LIN {X 0,Y 125.443,Z 652.418,A -85,B 0,C 180,E1 -25686.032,E2 -25686.032} C_VEL
LIN {X 0,Y 130.254,Z 643.589,A -85,B 0,C 180,E1 -25690.349,E2 -25690.349} C_VEL
LIN {X 0,Y 135.865,Z 633.156,A -85,B 0,C 180,E1 -25694.291,E2 -25694.291} C_VEL
LIN {X 0,Y 142.077,Z 620.726,A -85,B 0,C 180,E1 -25697.899,E2 -25697.899} C_VEL
LIN {X 0,Y 147.675,Z 608.285,A -85,B 0,C 180,E1 -25700.654,E2 -25700.654} C_VEL
LIN {X 0,Y 152.859,Z 595.068,A -85,B 0,C 180,E1 -25702.913,E2 -25702.913} C_VEL
LIN {X 0,Y 157.703,Z 580.518,A -85,B 0,C 180,E1 -25704.803,E2 -25704.803} C_VEL
LIN {X 0,Y 161.766,Z 565.791,A -85,B 0,C 180,E1 -25706.188,E2 -25706.188} C_VEL
LIN {X 0,Y 165,Z 549.941,A -85,B 0,C 180,E1 -25707.268,E2 -25707.268} C_VEL
LIN {X 0,Y 167.218,Z 532.789,A -85,B 0,C 180,E1 -25708.056,E2 -25708.056} C_VEL
LIN {X 0,Y 172.706,Z 478.21,A -85,B 0,C 180,E1 -25710.075,E2 -25710.075} C_VEL
LIN {X 0,Y 167.716,Z 464.569,A -85,B 0,C 180,E1 -25713.059,E2 -25713.059} C_VEL
LIN {X 0,Y 162.081,Z 450.718,A -85,B 0,C 180,E1 -25716.721,E2 -25716.721} C_VEL
LIN {X 0,Y 156.963,Z 439.698,A -85,B 0,C 180,E1 -25720.339,E2 -25720.339} C_VEL
LIN {X 0,Y 151.626,Z 431.129,A -85,B 0,C 180,E1 -25724.439,E2 -25724.439} C_VEL
LIN {X 0,Y 146.698,Z 423.586,A -85,B 0,C 180,E1 -25728.832,E2 -25728.832} C_VEL
LIN {X 0,Y 143.791,Z 419.372,A -85,B 0,C 180,E1 -25731.835,E2 -25731.835} C_VEL
LIN {X 0,Y 140.329,Z 414.378,A -85,B 0,C 180,E1 -25736.007,E2 -25736.007} C_VEL
LIN {X 0,Y 137.906,Z 411.663,A -85,B 0,C 180,E1 -25739.367,E2 -25739.367} C_VEL
LIN {X 0,Y 136.739,Z 409.178,A -85,B 0,C 180,E1 -25741.474,E2 -25741.474} C_VEL
LIN {X 0,Y 133.888,Z 406.923,A -85,B 0,C 180,E1 -25747.021,E2 -25747.021} C_VEL
LIN {X 0,Y 132.787,Z 404.232,A -85,B 0,C 180,E1 -25750.732,E2 -25750.732} C_VEL
LIN {X 0,Y 131.279,Z 403.638,A -85,B 0,C 180,E1 -25758.737,E2 -25758.737} C_VEL
LIN {X 0,Y 132.384,Z 404.128,A -85,B 0,C 180,E1 -25768.976,E2 -25768.976} C_VEL
LIN {X 0,Y 133.882,Z 407.624,A -85,B 0,C 180,E1 -25774.373,E2 -25774.373} C_VEL
LIN {X 0,Y 136.345,Z 409.759,A -85,B 0,C 180,E1 -25779.23,E2 -25779.23} C_VEL
LIN {X 0,Y 138.489,Z 413.228,A -85,B 0,C 180,E1 -25782.831,E2 -25782.831} C_VEL
LIN {X 0,Y 140.328,Z 415.144,A -85,B 0,C 180,E1 -25785.268,E2 -25785.268} C_VEL
LIN {X 0,Y 142.881,Z 418.739,A -85,B 0,C 180,E1 -25788.424,E2 -25788.424} C_VEL
LIN {X 0,Y 144.144,Z 420.426,A -85,B 0,C 180,E1 -25789.796,E2 -25789.796} C_VEL
LIN {X 0,Y 147.549,Z 425.18,A -85,B 0,C 180,E1 -25793.178,E2 -25793.178} C_VEL
LIN {X 0,Y 152.323,Z 432.249,A -85,B 0,C 180,E1 -25797.286,E2 -25797.286} C_VEL
LIN {X 0,Y 158.951,Z 442.925,A -85,B 0,C 180,E1 -25802.168,E2 -25802.168} C_VEL
LIN {X 0,Y 166.384,Z 455.969,A -85,B 0,C 180,E1 -25806.825,E2 -25806.825} C_VEL
LIN {X 0,Y 172.94,Z 469.275,A -85,B 0,C 180,E1 -25810.468,E2 -25810.468} C_VEL
LIN {X 0,Y 166.829,Z 528.834,A -85,B 0,C 180,E1 -25812.708,E2 -25812.708} C_VEL
LIN {X 0,Y 164.138,Z 544.967,A -85,B 0,C 180,E1 -25813.682,E2 -25813.682} C_VEL
LIN {X 0,Y 160.991,Z 559.376,A -85,B 0,C 180,E1 -25814.965,E2 -25814.965} C_VEL
LIN {X 0,Y 156.607,Z 574.603,A -85,B 0,C 180,E1 -25816.755,E2 -25816.755} C_VEL
LIN {X 0,Y 151.714,Z 588.809,A -85,B 0,C 180,E1 -25818.985,E2 -25818.985} C_VEL
LIN {X 0,Y 146.164,Z 602.31,A -85,B 0,C 180,E1 -25821.707,E2 -25821.707} C_VEL
LIN {X 0,Y 140.508,Z 614.537,A -85,B 0,C 180,E1 -25824.907,E2 -25824.907} C_VEL
LIN {X 0,Y 135.088,Z 625.294,A -85,B 0,C 180,E1 -25828.511,E2 -25828.511} C_VEL
LIN {X 0,Y 129.26,Z 635.988,A -85,B 0,C 180,E1 -25833.118,E2 -25833.118} C_VEL
LIN {X 0,Y 124.232,Z 644.963,A -85,B 0,C 180,E1 -25838.132,E2 -25838.132} C_VEL
LIN {X 0,Y 119.987,Z 652.541,A -85,B 0,C 180,E1 -25843.551,E2 -25843.551} C_VEL
LIN {X 0,Y 116.685,Z 658.822,A -85,B 0,C 180,E1 -25849.347,E2 -25849.347} C_VEL
LIN {X 0,Y 114.262,Z 664.018,A -85,B 0,C 180,E1 -25855.504,E2 -25855.504} C_VEL
LIN {X 0,Y 112.642,Z 668.237,A -85,B 0,C 180,E1 -25862.03,E2 -25862.03} C_VEL
LIN {X 0,Y 112.015,Z 671.471,A -85,B 0,C 180,E1 -25868.862,E2 -25868.862} C_VEL
LIN {X 0,Y 112.697,Z 673.827,A -85,B 0,C 180,E1 -25876.685,E2 -25876.685} C_VEL
LIN {X 0,Y 114.296,Z 674.743,A -85,B 0,C 180,E1 -25883.072,E2 -25883.072} C_VEL
LIN {X 0,Y 116.279,Z 674.886,A -85,B 0,C 180,E1 -25887.8,E2 -25887.8} C_VEL
LIN {X 0,Y 118.94,Z 674.527,A -85,B 0,C 180,E1 -25892.418,E2 -25892.418} C_VEL
LIN {X 0,Y 122.264,Z 673.586,A -85,B 0,C 180,E1 -25896.888,E2 -25896.888} C_VEL
LIN {X 0,Y 126.265,Z 672.105,A -85,B 0,C 180,E1 -25901.13,E2 -25901.13} C_VEL
LIN {X 0,Y 130.881,Z 670.075,A -85,B 0,C 180,E1 -25905.146,E2 -25905.146} C_VEL
LIN {X 0,Y 138.024,Z 666.375,A -85,B 0,C 180,E1 -25910.12,E2 -25910.12} C_VEL
LIN {X 0,Y 146.03,Z 661.626,A -85,B 0,C 180,E1 -25914.475,E2 -25914.475} C_VEL
LIN {X 0,Y 154.683,Z 655.759,A -85,B 0,C 180,E1 -25918.354,E2 -25918.354} C_VEL
LIN {X 0,Y 163.688,Z 648.719,A -85,B 0,C 180,E1 -25921.734,E2 -25921.734} C_VEL
LIN {X 0,Y 174.031,Z 639.5,A -85,B 0,C 180,E1 -25924.977,E2 -25924.977} C_VEL
LIN {X 0,Y 184.395,Z 628.842,A -85,B 0,C 180,E1 -25927.703,E2 -25927.703} C_VEL
LIN {X 0,Y 193.48,Z 617.944,A -85,B 0,C 180,E1 -25929.759,E2 -25929.759} C_VEL
LIN {X 0,Y 201.771,Z 606.367,A -85,B 0,C 180,E1 -25931.454,E2 -25931.454} C_VEL
LIN {X 0,Y 209.045,Z 594.538,A -85,B 0,C 180,E1 -25932.844,E2 -25932.844} C_VEL
LIN {X 0,Y 215.674,Z 581.801,A -85,B 0,C 180,E1 -25933.983,E2 -25933.983} C_VEL
LIN {X 0,Y 221.796,Z 567.365,A -85,B 0,C 180,E1 -25935.017,E2 -25935.017} C_VEL
LIN {X 0,Y 226.824,Z 552.153,A -85,B 0,C 180,E1 -25935.827,E2 -25935.827} C_VEL
LIN {X 0,Y 230.242,Z 538.347,A -85,B 0,C 180,E1 -25936.341,E2 -25936.341} C_VEL
LIN {X 0,Y 233.479,Z 518.913,A -85,B 0,C 180,E1 -25936.868,E2 -25936.868} C_VEL
LIN {X 0,Y 234.676,Z 510.745,A -85,B 0,C 180,E1 -25937.099,E2 -25937.099} C_VEL
LIN {X 0,Y 234.535,Z 509.573,A -85,B 0,C 180,E1 -25939.245,E2 -25939.245} C_VEL
LIN {X 0,Y 234.487,Z 510.416,A -85,B 0,C 180,E1 -25940.646,E2 -25940.646} C_VEL
LIN {X 0,Y 234.522,Z 512.099,A -85,B 0,C 180,E1 -25942.274,E2 -25942.274} C_VEL
LIN {X 0,Y 230.283,Z 538.9,A -85,B 0,C 180,E1 -25942.912,E2 -25942.912} C_VEL
LIN {X 0,Y 226.669,Z 553.893,A -85,B 0,C 180,E1 -25943.367,E2 -25943.367} C_VEL
LIN {X 0,Y 221.965,Z 568.306,A -85,B 0,C 180,E1 -25943.898,E2 -25943.898} C_VEL
LIN {X 0,Y 216.394,Z 581.875,A -85,B 0,C 180,E1 -25944.578,E2 -25944.578} C_VEL
LIN {X 0,Y 209.352,Z 595.9,A -85,B 0,C 180,E1 -25945.549,E2 -25945.549} C_VEL
LIN {X 0,Y 201.575,Z 608.795,A -85,B 0,C 180,E1 -25946.691,E2 -25946.691} C_VEL
LIN {X 0,Y 193.253,Z 620.7,A -85,B 0,C 180,E1 -25948.126,E2 -25948.126} C_VEL
LIN {X 0,Y 184.53,Z 631.604,A -85,B 0,C 180,E1 -25949.862,E2 -25949.862} C_VEL
LIN {X 0,Y 174.353,Z 642.657,A -85,B 0,C 180,E1 -25952.166,E2 -25952.166} C_VEL
LIN {X 0,Y 166.132,Z 650.629,A -85,B 0,C 180,E1 -25954.418,E2 -25954.418} C_VEL
LIN {X 0,Y 155.723,Z 659.68,A -85,B 0,C 180,E1 -25957.832,E2 -25957.832} C_VEL
LIN {X 0,Y 146.02,Z 667.142,A -85,B 0,C 180,E1 -25961.752,E2 -25961.752} C_VEL
LIN {X 0,Y 137.261,Z 673.246,A -85,B 0,C 180,E1 -25966.271,E2 -25966.271} C_VEL
LIN {X 0,Y 129.55,Z 678.069,A -85,B 0,C 180,E1 -25971.399,E2 -25971.399} C_VEL
LIN {X 0,Y 124.565,Z 680.957,A -85,B 0,C 180,E1 -25975.651,E2 -25975.651} C_VEL
LIN {X 0,Y 118.405,Z 684.199,A -85,B 0,C 180,E1 -25982.913,E2 -25982.913} C_VEL
LIN {X 0,Y 114.455,Z 685.901,A -85,B 0,C 180,E1 -25990.578,E2 -25990.578} C_VEL
LIN {X 0,Y 112.564,Z 686.363,A -85,B 0,C 180,E1 -25999.203,E2 -25999.203} C_VEL
LIN {X 0,Y 112.622,Z 685.531,A -85,B 0,C 180,E1 -26006.071,E2 -26006.071} C_VEL
LIN {X 0,Y 112.463,Z 685.102,A -85,B 0,C 180,E1 -26008.046,E2 -26008.046} C_VEL
LIN {X 0,Y 111.167,Z 684.151,A -85,B 0,C 180,E1 -26010.958,E2 -26010.958} C_VEL
LIN {X 0,Y 107.875,Z 681.964,A -85,B 0,C 180,E1 -26015.794,E2 -26015.794} C_VEL
LIN {X 0,Y 105.938,Z 679.776,A -85,B 0,C 180,E1 -26019.867,E2 -26019.867} C_VEL
LIN {X 0,Y 105.78,Z 678.569,A -85,B 0,C 180,E1 -26021.96,E2 -26021.96} C_VEL
LIN {X 0,Y 107.257,Z 673.673,A -85,B 0,C 180,E1 -26029.123,E2 -26029.123} C_VEL
LIN {X 0,Y 110.456,Z 666.96,A -85,B 0,C 180,E1 -26036.446,E2 -26036.446} C_VEL
LIN {X 0,Y 114.483,Z 659.638,A -85,B 0,C 180,E1 -26042.488,E2 -26042.488} C_VEL
LIN {X 0,Y 119.634,Z 650.778,A -85,B 0,C 180,E1 -26048.083,E2 -26048.083} C_VEL
LIN {X 0,Y 125.491,Z 640.608,A -85,B 0,C 180,E1 -26052.959,E2 -26052.959} C_VEL
LIN {X 0,Y 131.869,Z 629.081,A -85,B 0,C 180,E1 -26057.12,E2 -26057.12} C_VEL
LIN {X 0,Y 137.937,Z 617.091,A -85,B 0,C 180,E1 -26060.408,E2 -26060.408} C_VEL
LIN {X 0,Y 143.861,Z 604.032,A -85,B 0,C 180,E1 -26063.124,E2 -26063.124} C_VEL
LIN {X 0,Y 148.917,Z 590.956,A -85,B 0,C 180,E1 -26065.229,E2 -26065.229} C_VEL
LIN {X 0,Y 153.912,Z 575.773,A -85,B 0,C 180,E1 -26067.037,E2 -26067.037} C_VEL
LIN {X 0,Y 157.666,Z 561.167,A -85,B 0,C 180,E1 -26068.33,E2 -26068.33} C_VEL
LIN {X 0,Y 160.525,Z 546.659,A -85,B 0,C 180,E1 -26069.225,E2 -26069.225} C_VEL
LIN {X 0,Y 163.128,Z 525.318,A -85,B 0,C 180,E1 -26070.12,E2 -26070.12} C_VEL
LIN {X 0,Y 167.784,Z 480.393,A -85,B 0,C 180,E1 -26071.792,E2 -26071.792} C_VEL
LIN {X 0,Y 162.639,Z 466.125,A -85,B 0,C 180,E1 -26075.114,E2 -26075.114} C_VEL
LIN {X 0,Y 157.795,Z 454.04,A -85,B 0,C 180,E1 -26078.526,E2 -26078.526} C_VEL
LIN {X 0,Y 153.632,Z 444.809,A -85,B 0,C 180,E1 -26081.714,E2 -26081.714} C_VEL
LIN {X 0,Y 148.768,Z 436.819,A -85,B 0,C 180,E1 -26085.666,E2 -26085.666} C_VEL
LIN {X 0,Y 144.325,Z 429.702,A -85,B 0,C 180,E1 -26089.932,E2 -26089.932} C_VEL
LIN {X 0,Y 140.724,Z 424.449,A -85,B 0,C 180,E1 -26093.902,E2 -26093.902} C_VEL
LIN {X 0,Y 138.347,Z 420.857,A -85,B 0,C 180,E1 -26097.089,E2 -26097.089} C_VEL
LIN {X 0,Y 135.921,Z 417.683,A -85,B 0,C 180,E1 -26100.742,E2 -26100.742} C_VEL
LIN {X 0,Y 134.949,Z 415.845,A -85,B 0,C 180,E1 -26102.613,E2 -26102.613} C_VEL
LIN {X 0,Y 132.486,Z 413.636,A -85,B 0,C 180,E1 -26107.815,E2 -26107.815} C_VEL
LIN {X 0,Y 131.521,Z 411.063,A -85,B 0,C 180,E1 -26111.469,E2 -26111.469} C_VEL
LIN {X 0,Y 130.217,Z 410.646,A -85,B 0,C 180,E1 -26118.896,E2 -26118.896} C_VEL
LIN {X 0,Y 131.207,Z 411.194,A -85,B 0,C 180,E1 -26128.624,E2 -26128.624} C_VEL
LIN {X 0,Y 132.618,Z 414.564,A -85,B 0,C 180,E1 -26133.958,E2 -26133.958} C_VEL
LIN {X 0,Y 134.853,Z 416.661,A -85,B 0,C 180,E1 -26138.582,E2 -26138.582} C_VEL
LIN {X 0,Y 137.334,Z 420.474,A -85,B 0,C 180,E1 -26142.835,E2 -26142.835} C_VEL
LIN {X 0,Y 138.514,Z 421.759,A -85,B 0,C 180,E1 -26144.428,E2 -26144.428} C_VEL
LIN {X 0,Y 141.317,Z 425.66,A -85,B 0,C 180,E1 -26148.022,E2 -26148.022} C_VEL
LIN {X 0,Y 145.536,Z 431.898,A -85,B 0,C 180,E1 -26152.495,E2 -26152.495} C_VEL
LIN {X 0,Y 150.085,Z 439.007,A -85,B 0,C 180,E1 -26156.614,E2 -26156.614} C_VEL
LIN {X 0,Y 155.769,Z 448.442,A -85,B 0,C 180,E1 -26161.007,E2 -26161.007} C_VEL
LIN {X 0,Y 162.755,Z 461.017,A -85,B 0,C 180,E1 -26165.629,E2 -26165.629} C_VEL
LIN {X 0,Y 167.887,Z 471.772,A -85,B 0,C 180,E1 -26168.716,E2 -26168.716} C_VEL
LIN {X 0,Y 161.747,Z 530.169,A -85,B 0,C 180,E1 -26170.982,E2 -26170.982} C_VEL
LIN {X 0,Y 158.973,Z 546.096,A -85,B 0,C 180,E1 -26171.974,E2 -26171.974} C_VEL
LIN {X 0,Y 155.68,Z 560.439,A -85,B 0,C 180,E1 -26173.275,E2 -26173.275} C_VEL
LIN {X 0,Y 151.202,Z 575.356,A -85,B 0,C 180,E1 -26175.052,E2 -26175.052} C_VEL
LIN {X 0,Y 146.407,Z 588.792,A -85,B 0,C 180,E1 -26177.174,E2 -26177.174} C_VEL
LIN {X 0,Y 140.636,Z 602.367,A -85,B 0,C 180,E1 -26179.928,E2 -26179.928} C_VEL
LIN {X 0,Y 135.123,Z 613.933,A -85,B 0,C 180,E1 -26182.966,E2 -26182.966} C_VEL
LIN {X 0,Y 129.08,Z 625.454,A -85,B 0,C 180,E1 -26186.88,E2 -26186.88} C_VEL
LIN {X 0,Y 122.957,Z 636.197,A -85,B 0,C 180,E1 -26191.639,E2 -26191.639} C_VEL
LIN {X 0,Y 117.675,Z 645.207,A -85,B 0,C 180,E1 -26196.862,E2 -26196.862} C_VEL
LIN {X 0,Y 113.197,Z 652.811,A -85,B 0,C 180,E1 -26202.55,E2 -26202.55} C_VEL
LIN {X 0,Y 109.698,Z 659.129,A -85,B 0,C 180,E1 -26208.685,E2 -26208.685} C_VEL
LIN {X 0,Y 107.066,Z 664.573,A -85,B 0,C 180,E1 -26215.542,E2 -26215.542} C_VEL
LIN {X 0,Y 105.494,Z 668.604,A -85,B 0,C 180,E1 -26222.208,E2 -26222.208} C_VEL
LIN {X 0,Y 104.977,Z 670.854,A -85,B 0,C 180,E1 -26227.053,E2 -26227.053} C_VEL
LIN {X 0,Y 105.069,Z 672.861,A -85,B 0,C 180,E1 -26232.624,E2 -26232.624} C_VEL
LIN {X 0,Y 105.895,Z 674.344,A -85,B 0,C 180,E1 -26238.417,E2 -26238.417} C_VEL
LIN {X 0,Y 108.714,Z 675.345,A -85,B 0,C 180,E1 -26247.186,E2 -26247.186} C_VEL
LIN {X 0,Y 112.612,Z 675.038,A -85,B 0,C 180,E1 -26254.095,E2 -26254.095} C_VEL
LIN {X 0,Y 118.688,Z 673.438,A -85,B 0,C 180,E1 -26261.343,E2 -26261.343} C_VEL
LIN {X 0,Y 125.217,Z 670.937,A -85,B 0,C 180,E1 -26267.025,E2 -26267.025} C_VEL
LIN {X 0,Y 134.515,Z 666.518,A -85,B 0,C 180,E1 -26273.078,E2 -26273.078} C_VEL
LIN {X 0,Y 142.64,Z 661.967,A -85,B 0,C 180,E1 -26277.175,E2 -26277.175} C_VEL
LIN {X 0,Y 152.31,Z 655.695,A -85,B 0,C 180,E1 -26281.144,E2 -26281.144} C_VEL
LIN {X 0,Y 163.472,Z 647.228,A -85,B 0,C 180,E1 -26284.932,E2 -26284.932} C_VEL
LIN {X 0,Y 172.952,Z 638.972,A -85,B 0,C 180,E1 -26287.579,E2 -26287.579} C_VEL
LIN {X 0,Y 182.825,Z 629.028,A -85,B 0,C 180,E1 -26289.962,E2 -26289.962} C_VEL
LIN {X 0,Y 193.039,Z 617.073,A -85,B 0,C 180,E1 -26292.084,E2 -26292.084} C_VEL
LIN {X 0,Y 202.022,Z 604.652,A -85,B 0,C 180,E1 -26293.754,E2 -26293.754} C_VEL
LIN {X 0,Y 209.631,Z 592.193,A -85,B 0,C 180,E1 -26295.06,E2 -26295.06} C_VEL
LIN {X 0,Y 216.539,Z 578.673,A -85,B 0,C 180,E1 -26296.136,E2 -26296.136} C_VEL
LIN {X 0,Y 222.493,Z 564.251,A -85,B 0,C 180,E1 -26297.053,E2 -26297.053} C_VEL
LIN {X 0,Y 227.283,Z 549.222,A -85,B 0,C 180,E1 -26297.747,E2 -26297.747} C_VEL
LIN {X 0,Y 230.679,Z 534.54,A -85,B 0,C 180,E1 -26298.228,E2 -26298.228} C_VEL
LIN {X 0,Y 233.474,Z 516.829,A -85,B 0,C 180,E1 -26298.706,E2 -26298.706} C_VEL
LIN {X 0,Y 233.429,Z 516.847,A -85,B 0,C 180,E1 -26299.852,E2 -26299.852} C_VEL
LIN {X 0,Y 233.346,Z 517.898,A -85,B 0,C 180,E1 -26300.673,E2 -26300.673} C_VEL
LIN {X 0,Y 229.749,Z 539.399,A -85,B 0,C 180,E1 -26301.155,E2 -26301.155} C_VEL
LIN {X 0,Y 226.011,Z 554.187,A -85,B 0,C 180,E1 -26301.569,E2 -26301.569} C_VEL
LIN {X 0,Y 220.922,Z 569.123,A -85,B 0,C 180,E1 -26302.098,E2 -26302.098} C_VEL
LIN {X 0,Y 214.446,Z 584.005,A -85,B 0,C 180,E1 -26302.817,E2 -26302.817} C_VEL
LIN {X 0,Y 206.485,Z 598.908,A -85,B 0,C 180,E1 -26303.831,E2 -26303.831} C_VEL
LIN {X 0,Y 198.573,Z 611.266,A -85,B 0,C 180,E1 -26304.913,E2 -26304.913} C_VEL
LIN {X 0,Y 190.092,Z 622.713,A -85,B 0,C 180,E1 -26306.288,E2 -26306.288} C_VEL
LIN {X 0,Y 180.914,Z 633.504,A -85,B 0,C 180,E1 -26308.014,E2 -26308.014} C_VEL
LIN {X 0,Y 170.738,Z 643.947,A -85,B 0,C 180,E1 -26310.183,E2 -26310.183} C_VEL
LIN {X 0,Y 162.261,Z 651.629,A -85,B 0,C 180,E1 -26312.369,E2 -26312.369} C_VEL
LIN {X 0,Y 151.49,Z 660.357,A -85,B 0,C 180,E1 -26315.719,E2 -26315.719} C_VEL
LIN {X 0,Y 141.39,Z 667.603,A -85,B 0,C 180,E1 -26319.604,E2 -26319.604} C_VEL
LIN {X 0,Y 132.207,Z 673.487,A -85,B 0,C 180,E1 -26324.138,E2 -26324.138} C_VEL
LIN {X 0,Y 124.046,Z 678.181,A -85,B 0,C 180,E1 -26329.34,E2 -26329.34} C_VEL
LIN {X 0,Y 115.608,Z 682.412,A -85,B 0,C 180,E1 -26336.828,E2 -26336.828} C_VEL
LIN {X 0,Y 110.577,Z 684.609,A -85,B 0,C 180,E1 -26343.581,E2 -26343.581} C_VEL
LIN {X 0,Y 107.152,Z 685.729,A -85,B 0,C 180,E1 -26350.854,E2 -26350.854} C_VEL
LIN {X 0,Y 105.539,Z 685.831,A -85,B 0,C 180,E1 -26358.475,E2 -26358.475} C_VEL
LIN {X 0,Y 105.602,Z 684.778,A -85,B 0,C 180,E1 -26366.612,E2 -26366.612} C_VEL
LIN {X 0,Y 105.869,Z 683.919,A -85,B 0,C 180,E1 -26369.998,E2 -26369.998} C_VEL
LIN {X 0,Y 105.61,Z 682.57,A -85,B 0,C 180,E1 -26373.814,E2 -26373.814} C_VEL
LIN {X 0,Y 105.78,Z 678.569,A -85,B 0,C 180,E1 -26381.96,E2 -26381.96} C_VEL
LIN {X 0,Y 105.56,Z 676.657,A -85,B 0,C 180,E1 -26384.983,E2 -26384.983} C_VEL
LIN {X 0,Y 103.95,Z 673.014,A -85,B 0,C 180,E1 -26389.951,E2 -26389.951} C_VEL
LIN {X 0,Y 103.009,Z 668.889,A -85,B 0,C 180,E1 -26394.937,E2 -26394.937} C_VEL
LIN {X 0,Y 103.837,Z 666.115,A -85,B 0,C 180,E1 -26397.83,E2 -26397.83} C_VEL
LIN {X 0,Y 108.471,Z 658.224,A -85,B 0,C 180,E1 -26404.534,E2 -26404.534} C_VEL
LIN {X 0,Y 114.042,Z 649.151,A -85,B 0,C 180,E1 -26410.319,E2 -26410.319} C_VEL
LIN {X 0,Y 119.655,Z 639.871,A -85,B 0,C 180,E1 -26414.813,E2 -26414.813} C_VEL
LIN {X 0,Y 125.971,Z 628.919,A -85,B 0,C 180,E1 -26418.864,E2 -26418.864} C_VEL
LIN {X 0,Y 132.281,Z 616.978,A -85,B 0,C 180,E1 -26422.211,E2 -26422.211} C_VEL
LIN {X 0,Y 138.4,Z 603.968,A -85,B 0,C 180,E1 -26424.966,E2 -26424.966} C_VEL
LIN {X 0,Y 144.13,Z 589.609,A -85,B 0,C 180,E1 -26427.271,E2 -26427.271} C_VEL
LIN {X 0,Y 149.116,Z 574.796,A -85,B 0,C 180,E1 -26429.001,E2 -26429.001} C_VEL
LIN {X 0,Y 152.989,Z 560.013,A -85,B 0,C 180,E1 -26430.284,E2 -26430.284} C_VEL
LIN {X 0,Y 155.918,Z 545.163,A -85,B 0,C 180,E1 -26431.178,E2 -26431.178} C_VEL
LIN {X 0,Y 158.783,Z 521.467,A -85,B 0,C 180,E1 -26432.148,E2 -26432.148} C_VEL
LIN {X 0,Y 162.917,Z 482.399,A -85,B 0,C 180,E1 -26433.623,E2 -26433.623} C_VEL
LIN {X 0,Y 158.002,Z 468.529,A -85,B 0,C 180,E1 -26437.096,E2 -26437.096} C_VEL
LIN {X 0,Y 153.53,Z 457.117,A -85,B 0,C 180,E1 -26440.506,E2 -26440.506} C_VEL
LIN {X 0,Y 150.255,Z 449.629,A -85,B 0,C 180,E1 -26443.267,E2 -26443.267} C_VEL
LIN {X 0,Y 145.361,Z 441.499,A -85,B 0,C 180,E1 -26447.529,E2 -26447.529} C_VEL
LIN {X 0,Y 141.711,Z 435.491,A -85,B 0,C 180,E1 -26451.312,E2 -26451.312} C_VEL
LIN {X 0,Y 138.685,Z 430.781,A -85,B 0,C 180,E1 -26454.927,E2 -26454.927} C_VEL
LIN {X 0,Y 136.47,Z 427.366,A -85,B 0,C 180,E1 -26458.061,E2 -26458.061} C_VEL
LIN {X 0,Y 134.107,Z 423.941,A -85,B 0,C 180,E1 -26461.948,E2 -26461.948} C_VEL
LIN {X 0,Y 133.619,Z 422.763,A -85,B 0,C 180,E1 -26463.016,E2 -26463.016} C_VEL
LIN {X 0,Y 131.176,Z 420.479,A -85,B 0,C 180,E1 -26468.412,E2 -26468.412} C_VEL
LIN {X 0,Y 130.308,Z 418.034,A -85,B 0,C 180,E1 -26472.018,E2 -26472.018} C_VEL
LIN {X 0,Y 129.156,Z 417.648,A -85,B 0,C 180,E1 -26479.057,E2 -26479.057} C_VEL
LIN {X 0,Y 129.999,Z 418.074,A -85,B 0,C 180,E1 -26488.051,E2 -26488.051} C_VEL
LIN {X 0,Y 131.238,Z 421.311,A -85,B 0,C 180,E1 -26493.207,E2 -26493.207} C_VEL
LIN {X 0,Y 133.37,Z 423.464,A -85,B 0,C 180,E1 -26497.889,E2 -26497.889} C_VEL
LIN {X 0,Y 135.799,Z 427.282,A -85,B 0,C 180,E1 -26502.284,E2 -26502.284} C_VEL
LIN {X 0,Y 136.813,Z 428.55,A -85,B 0,C 180,E1 -26503.747,E2 -26503.747} C_VEL
LIN {X 0,Y 139.927,Z 433.152,A -85,B 0,C 180,E1 -26507.863,E2 -26507.863} C_VEL
LIN {X 0,Y 142.896,Z 437.627,A -85,B 0,C 180,E1 -26511.152,E2 -26511.152} C_VEL
LIN {X 0,Y 147.126,Z 444.413,A -85,B 0,C 180,E1 -26515.253,E2 -26515.253} C_VEL
LIN {X 0,Y 152.516,Z 453.675,A -85,B 0,C 180,E1 -26519.688,E2 -26519.688} C_VEL
LIN {X 0,Y 159.282,Z 466.268,A -85,B 0,C 180,E1 -26524.462,E2 -26524.462} C_VEL
LIN {X 0,Y 163.129,Z 474.725,A -85,B 0,C 180,E1 -26526.959,E2 -26526.959} C_VEL
LIN {X 0,Y 156.967,Z 530.563,A -85,B 0,C 180,E1 -26529.098,E2 -26529.098} C_VEL
LIN {X 0,Y 154.107,Z 546.473,A -85,B 0,C 180,E1 -26530.087,E2 -26530.087} C_VEL
LIN {X 0,Y 150.582,Z 561.25,A -85,B 0,C 180,E1 -26531.44,E2 -26531.44} C_VEL
LIN {X 0,Y 145.97,Z 576.02,A -85,B 0,C 180,E1 -26533.21,E2 -26533.21} C_VEL
LIN {X 0,Y 140.572,Z 590.392,A -85,B 0,C 180,E1 -26535.525,E2 -26535.525} C_VEL
LIN {X 0,Y 134.632,Z 603.748,A -85,B 0,C 180,E1 -26538.331,E2 -26538.331} C_VEL
LIN {X 0,Y 128.457,Z 615.986,A -85,B 0,C 180,E1 -26541.701,E2 -26541.701} C_VEL
LIN {X 0,Y 122.049,Z 627.519,A -85,B 0,C 180,E1 -26545.874,E2 -26545.874} C_VEL
LIN {X 0,Y 115.784,Z 637.984,A -85,B 0,C 180,E1 -26550.871,E2 -26550.871} C_VEL
LIN {X 0,Y 110.319,Z 646.77,A -85,B 0,C 180,E1 -26556.403,E2 -26556.403} C_VEL
LIN {X 0,Y 105.756,Z 654.177,A -85,B 0,C 180,E1 -26562.475,E2 -26562.475} C_VEL
LIN {X 0,Y 102.446,Z 659.971,A -85,B 0,C 180,E1 -26568.586,E2 -26568.586} C_VEL
LIN {X 0,Y 100.055,Z 664.657,A -85,B 0,C 180,E1 -26574.928,E2 -26574.928} C_VEL
LIN {X 0,Y 98.534,Z 668.314,A -85,B 0,C 180,E1 -26581.136,E2 -26581.136} C_VEL
LIN {X 0,Y 97.857,Z 672.22,A -85,B 0,C 180,E1 -26590.271,E2 -26590.271} C_VEL
LIN {X 0,Y 98.276,Z 673.825,A -85,B 0,C 180,E1 -26595.656,E2 -26595.656} C_VEL
LIN {X 0,Y 99.346,Z 674.959,A -85,B 0,C 180,E1 -26601.096,E2 -26601.096} C_VEL
LIN {X 0,Y 101.136,Z 675.62,A -85,B 0,C 180,E1 -26606.503,E2 -26606.503} C_VEL
LIN {X 0,Y 103.713,Z 675.796,A -85,B 0,C 180,E1 -26611.758,E2 -26611.758} C_VEL
LIN {X 0,Y 107.027,Z 675.479,A -85,B 0,C 180,E1 -26616.831,E2 -26616.831} C_VEL
LIN {X 0,Y 111.096,Z 674.608,A -85,B 0,C 180,E1 -26621.611,E2 -26621.611} C_VEL
LIN {X 0,Y 115.865,Z 673.176,A -85,B 0,C 180,E1 -26626.056,E2 -26626.056} C_VEL
LIN {X 0,Y 123.924,Z 670.14,A -85,B 0,C 180,E1 -26631.938,E2 -26631.938} C_VEL
LIN {X 0,Y 133.678,Z 665.542,A -85,B 0,C 180,E1 -26637.345,E2 -26637.345} C_VEL
LIN {X 0,Y 143.576,Z 660.015,A -85,B 0,C 180,E1 -26641.596,E2 -26641.596} C_VEL
LIN {X 0,Y 153.983,Z 653.188,A -85,B 0,C 180,E1 -26645.236,E2 -26645.236} C_VEL
LIN {X 0,Y 164.03,Z 645.513,A -85,B 0,C 180,E1 -26648.157,E2 -26648.157} C_VEL
LIN {X 0,Y 174.404,Z 636.427,A -85,B 0,C 180,E1 -26650.711,E2 -26650.711} C_VEL
LIN {X 0,Y 183.69,Z 627.048,A -85,B 0,C 180,E1 -26652.672,E2 -26652.672} C_VEL
LIN {X 0,Y 193.31,Z 615.759,A -85,B 0,C 180,E1 -26654.474,E2 -26654.474} C_VEL
LIN {X 0,Y 202.907,Z 602.498,A -85,B 0,C 180,E1 -26656.086,E2 -26656.086} C_VEL
LIN {X 0,Y 210.147,Z 590.614,A -85,B 0,C 180,E1 -26657.181,E2 -26657.181} C_VEL
LIN {X 0,Y 216.8,Z 577.54,A -85,B 0,C 180,E1 -26658.126,E2 -26658.126} C_VEL
LIN {X 0,Y 222.435,Z 563.889,A -85,B 0,C 180,E1 -26658.931,E2 -26658.931} C_VEL
LIN {X 0,Y 227.167,Z 549.161,A -85,B 0,C 180,E1 -26659.561,E2 -26659.561} C_VEL
LIN {X 0,Y 223.413,Z 561.311,A -85,B 0,C 180,E1 -26659.981,E2 -26659.981} C_VEL
LIN {X 0,Y 217.631,Z 576.045,A -85,B 0,C 180,E1 -26660.526,E2 -26660.526} C_VEL
LIN {X 0,Y 211.097,Z 589.484,A -85,B 0,C 180,E1 -26661.218,E2 -26661.218} C_VEL
LIN {X 0,Y 202.994,Z 603.24,A -85,B 0,C 180,E1 -26662.159,E2 -26662.159} C_VEL
LIN {X 0,Y 194.193,Z 615.824,A -85,B 0,C 180,E1 -26663.313,E2 -26663.313} C_VEL
LIN {X 0,Y 184.491,Z 627.797,A -85,B 0,C 180,E1 -26664.84,E2 -26664.84} C_VEL
LIN {X 0,Y 174.86,Z 638.081,A -85,B 0,C 180,E1 -26666.582,E2 -26666.582} C_VEL
LIN {X 0,Y 164.443,Z 647.746,A -85,B 0,C 180,E1 -26668.819,E2 -26668.819} C_VEL
LIN {X 0,Y 158.609,Z 652.649,A -85,B 0,C 180,E1 -26670.224,E2 -26670.224} C_VEL
LIN {X 0,Y 147.482,Z 661.121,A -85,B 0,C 180,E1 -26673.493,E2 -26673.493} C_VEL
LIN {X 0,Y 136.984,Z 668.075,A -85,B 0,C 180,E1 -26677.321,E2 -26677.321} C_VEL
LIN {X 0,Y 127.356,Z 673.75,A -85,B 0,C 180,E1 -26681.84,E2 -26681.84} C_VEL
LIN {X 0,Y 120.795,Z 677.242,A -85,B 0,C 180,E1 -26685.717,E2 -26685.717} C_VEL
LIN {X 0,Y 113.018,Z 680.858,A -85,B 0,C 180,E1 -26691.547,E2 -26691.547} C_VEL
LIN {X 0,Y 106.734,Z 683.441,A -85,B 0,C 180,E1 -26698.211,E2 -26698.211} C_VEL
LIN {X 0,Y 102.069,Z 684.993,A -85,B 0,C 180,E1 -26705.596,E2 -26705.596} C_VEL
LIN {X 0,Y 99.245,Z 685.451,A -85,B 0,C 180,E1 -26713.543,E2 -26713.543} C_VEL
LIN {X 0,Y 98.298,Z 684.884,A -85,B 0,C 180,E1 -26721.777,E2 -26721.777} C_VEL
LIN {X 0,Y 98.55,Z 684.016,A -85,B 0,C 180,E1 -26726.734,E2 -26726.734} C_VEL
LIN {X 0,Y 98.805,Z 683.221,A -85,B 0,C 180,E1 -26729.998,E2 -26729.998} C_VEL
LIN {X 0,Y 98.516,Z 681.822,A -85,B 0,C 180,E1 -26734.089,E2 -26734.089} C_VEL
LIN {X 0,Y 98.751,Z 677.956,A -85,B 0,C 180,E1 -26742.326,E2 -26742.326} C_VEL
LIN {X 0,Y 100.513,Z 672.627,A -85,B 0,C 180,E1 -26750.461,E2 -26750.461} C_VEL
LIN {X 0,Y 103.837,Z 666.115,A -85,B 0,C 180,E1 -26757.83,E2 -26757.83} C_VEL
LIN {X 0,Y 104.86,Z 663.251,A -85,B 0,C 180,E1 -26760.612,E2 -26760.612} C_VEL
LIN {X 0,Y 105.202,Z 658.074,A -85,B 0,C 180,E1 -26765.228,E2 -26765.228} C_VEL
LIN {X 0,Y 106.025,Z 652.475,A -85,B 0,C 180,E1 -26769.654,E2 -26769.654} C_VEL
LIN {X 0,Y 107.743,Z 648.816,A -85,B 0,C 180,E1 -26772.004,E2 -26772.004} C_VEL
LIN {X 0,Y 113.609,Z 639.629,A -85,B 0,C 180,E1 -26776.622,E2 -26776.622} C_VEL
LIN {X 0,Y 120.19,Z 628.716,A -85,B 0,C 180,E1 -26780.783,E2 -26780.783} C_VEL
LIN {X 0,Y 126.754,Z 616.831,A -85,B 0,C 180,E1 -26784.181,E2 -26784.181} C_VEL
LIN {X 0,Y 133.093,Z 603.893,A -85,B 0,C 180,E1 -26786.957,E2 -26786.957} C_VEL
LIN {X 0,Y 139.016,Z 589.668,A -85,B 0,C 180,E1 -26789.251,E2 -26789.251} C_VEL
LIN {X 0,Y 144.103,Z 575.067,A -85,B 0,C 180,E1 -26790.97,E2 -26790.97} C_VEL
LIN {X 0,Y 148.136,Z 560.286,A -85,B 0,C 180,E1 -26792.262,E2 -26792.262} C_VEL
LIN {X 0,Y 151.114,Z 545.995,A -85,B 0,C 180,E1 -26793.126,E2 -26793.126} C_VEL
LIN {X 0,Y 153.884,Z 524.679,A -85,B 0,C 180,E1 -26794.012,E2 -26794.012} C_VEL
LIN {X 0,Y 158.324,Z 484.902,A -85,B 0,C 180,E1 -26795.474,E2 -26795.474} C_VEL
LIN {X 0,Y 153.987,Z 472.299,A -85,B 0,C 180,E1 -26798.763,E2 -26798.763} C_VEL
LIN {X 0,Y 150.016,Z 461.686,A -85,B 0,C 180,E1 -26802.093,E2 -26802.093} C_VEL
LIN {X 0,Y 147.114,Z 454.892,A -85,B 0,C 180,E1 -26804.673,E2 -26804.673} C_VEL
LIN {X 0,Y 141.689,Z 445.281,A -85,B 0,C 180,E1 -26809.958,E2 -26809.958} C_VEL
LIN {X 0,Y 138.167,Z 439.69,A -85,B 0,C 180,E1 -26813.966,E2 -26813.966} C_VEL
LIN {X 0,Y 136.54,Z 436.874,A -85,B 0,C 180,E1 -26816.198,E2 -26816.198} C_VEL
LIN {X 0,Y 134.712,Z 433.959,A -85,B 0,C 180,E1 -26818.917,E2 -26818.917} C_VEL
LIN {X 0,Y 132.415,Z 430.348,A -85,B 0,C 180,E1 -26823.044,E2 -26823.044} C_VEL
LIN {X 0,Y 131.953,Z 429.486,A -85,B 0,C 180,E1 -26824.079,E2 -26824.079} C_VEL
LIN {X 0,Y 129.695,Z 426.959,A -85,B 0,C 180,E1 -26829.641,E2 -26829.641} C_VEL
LIN {X 0,Y 129.102,Z 424.981,A -85,B 0,C 180,E1 -26832.578,E2 -26832.578} C_VEL
LIN {X 0,Y 128.108,Z 424.783,A -85,B 0,C 180,E1 -26842.584,E2 -26842.584} C_VEL
LIN {X 0,Y 128.839,Z 425.218,A -85,B 0,C 180,E1 -26847.792,E2 -26847.792} C_VEL
LIN {X 0,Y 129.975,Z 428.21,A -85,B 0,C 180,E1 -26852.734,E2 -26852.734} C_VEL
LIN {X 0,Y 131.87,Z 430.272,A -85,B 0,C 180,E1 -26857.135,E2 -26857.135} C_VEL
LIN {X 0,Y 134.554,Z 434.345,A -85,B 0,C 180,E1 -26862.133,E2 -26862.133} C_VEL
LIN {X 0,Y 137.93,Z 439.576,A -85,B 0,C 180,E1 -26866.919,E2 -26866.919} C_VEL
LIN {X 0,Y 141.248,Z 444.837,A -85,B 0,C 180,E1 -26870.788,E2 -26870.788} C_VEL
LIN {X 0,Y 145.274,Z 451.704,A -85,B 0,C 180,E1 -26874.829,E2 -26874.829} C_VEL
LIN {X 0,Y 150.049,Z 460.284,A -85,B 0,C 180,E1 -26878.912,E2 -26878.912} C_VEL
LIN {X 0,Y 155.98,Z 471.848,A -85,B 0,C 180,E1 -26883.361,E2 -26883.361} C_VEL
LIN {X 0,Y 158.476,Z 477.549,A -85,B 0,C 180,E1 -26885.082,E2 -26885.082} C_VEL
LIN {X 0,Y 152.376,Z 530.74,A -85,B 0,C 180,E1 -26887.098,E2 -26887.098} C_VEL
LIN {X 0,Y 149.577,Z 545.936,A -85,B 0,C 180,E1 -26888.013,E2 -26888.013} C_VEL
LIN {X 0,Y 145.91,Z 561.037,A -85,B 0,C 180,E1 -26889.378,E2 -26889.378} C_VEL
LIN {X 0,Y 141.099,Z 576.008,A -85,B 0,C 180,E1 -26891.154,E2 -26891.154} C_VEL
LIN {X 0,Y 135.574,Z 590.259,A -85,B 0,C 180,E1 -26893.436,E2 -26893.436} C_VEL
LIN {X 0,Y 130.084,Z 602.286,A -85,B 0,C 180,E1 -26895.906,E2 -26895.906} C_VEL
LIN {X 0,Y 123.515,Z 614.989,A -85,B 0,C 180,E1 -26899.345,E2 -26899.345} C_VEL
LIN {X 0,Y 117.414,Z 625.672,A -85,B 0,C 180,E1 -26903.126,E2 -26903.126} C_VEL
LIN {X 0,Y 110.899,Z 636.17,A -85,B 0,C 180,E1 -26908.004,E2 -26908.004} C_VEL
LIN {X 0,Y 104.779,Z 645.587,A -85,B 0,C 180,E1 -26913.848,E2 -26913.848} C_VEL
LIN {X 0,Y 99.178,Z 654.131,A -85,B 0,C 180,E1 -26920.997,E2 -26920.997} C_VEL
LIN {X 0,Y 95.697,Z 659.828,A -85,B 0,C 180,E1 -26927.302,E2 -26927.302} C_VEL
LIN {X 0,Y 92.893,Z 665.073,A -85,B 0,C 180,E1 -26934.781,E2 -26934.781} C_VEL
LIN {X 0,Y 91.174,Z 669.281,A -85,B 0,C 180,E1 -26942.658,E2 -26942.658} C_VEL
LIN {X 0,Y 90.728,Z 671.904,A -85,B 0,C 180,E1 -26949.227,E2 -26949.227} C_VEL
LIN {X 0,Y 91.229,Z 674.001,A -85,B 0,C 180,E1 -26956.103,E2 -26956.103} C_VEL
LIN {X 0,Y 93.557,Z 675.794,A -85,B 0,C 180,E1 -26965.726,E2 -26965.726} C_VEL
LIN {X 0,Y 97.857,Z 676.255,A -85,B 0,C 180,E1 -26974.473,E2 -26974.473} C_VEL
LIN {X 0,Y 103.498,Z 675.586,A -85,B 0,C 180,E1 -26981.932,E2 -26981.932} C_VEL
LIN {X 0,Y 111.335,Z 673.647,A -85,B 0,C 180,E1 -26989.082,E2 -26989.082} C_VEL
LIN {X 0,Y 119.952,Z 670.649,A -85,B 0,C 180,E1 -26994.907,E2 -26994.907} C_VEL
LIN {X 0,Y 129.879,Z 666.343,A -85,B 0,C 180,E1 -26999.999,E2 -26999.999} C_VEL
LIN {X 0,Y 140.978,Z 660.498,A -85,B 0,C 180,E1 -27004.398,E2 -27004.398} C_VEL
LIN {X 0,Y 152.078,Z 653.525,A -85,B 0,C 180,E1 -27007.968,E2 -27007.968} C_VEL
LIN {X 0,Y 162.868,Z 645.622,A -85,B 0,C 180,E1 -27010.812,E2 -27010.812} C_VEL
LIN {X 0,Y 174.18,Z 635.942,A -85,B 0,C 180,E1 -27013.317,E2 -27013.317} C_VEL
LIN {X 0,Y 185.3,Z 624.767,A -85,B 0,C 180,E1 -27015.396,E2 -27015.396} C_VEL
LIN {X 0,Y 194.89,Z 613.434,A -85,B 0,C 180,E1 -27016.954,E2 -27016.954} C_VEL
LIN {X 0,Y 204.234,Z 600.32,A -85,B 0,C 180,E1 -27018.377,E2 -27018.377} C_VEL
LIN {X 0,Y 209.409,Z 591.807,A -85,B 0,C 180,E1 -27019.079,E2 -27019.079} C_VEL
LIN {X 0,Y 208.74,Z 593.059,A -85,B 0,C 180,E1 -27019.484,E2 -27019.484} C_VEL
LIN {X 0,Y 200.514,Z 606.142,A -85,B 0,C 180,E1 -27020.348,E2 -27020.348} C_VEL
LIN {X 0,Y 191.583,Z 618.174,A -85,B 0,C 180,E1 -27021.429,E2 -27021.429} C_VEL
LIN {X 0,Y 181.508,Z 629.818,A -85,B 0,C 180,E1 -27022.896,E2 -27022.896} C_VEL
LIN {X 0,Y 170.294,Z 640.966,A -85,B 0,C 180,E1 -27024.776,E2 -27024.776} C_VEL
LIN {X 0,Y 159.659,Z 650.135,A -85,B 0,C 180,E1 -27026.951,E2 -27026.951} C_VEL
LIN {X 0,Y 150.873,Z 656.897,A -85,B 0,C 180,E1 -27029.14,E2 -27029.14} C_VEL
LIN {X 0,Y 138.184,Z 665.382,A -85,B 0,C 180,E1 -27032.944,E2 -27032.944} C_VEL
LIN {X 0,Y 127.657,Z 671.472,A -85,B 0,C 180,E1 -27037.034,E2 -27037.034} C_VEL
LIN {X 0,Y 115.793,Z 677.374,A -85,B 0,C 180,E1 -27043.251,E2 -27043.251} C_VEL
LIN {X 0,Y 107.495,Z 680.84,A -85,B 0,C 180,E1 -27049.169,E2 -27049.169} C_VEL
LIN {X 0,Y 100.718,Z 683.228,A -85,B 0,C 180,E1 -27056.064,E2 -27056.064} C_VEL
LIN {X 0,Y 95.577,Z 684.628,A -85,B 0,C 180,E1 -27063.818,E2 -27063.818} C_VEL
LIN {X 0,Y 92.388,Z 684.991,A -85,B 0,C 180,E1 -27072.283,E2 -27072.283} C_VEL
LIN {X 0,Y 91.242,Z 684.276,A -85,B 0,C 180,E1 -27081.136,E2 -27081.136} C_VEL
LIN {X 0,Y 91.505,Z 683.27,A -85,B 0,C 180,E1 -27086.796,E2 -27086.796} C_VEL
LIN {X 0,Y 91.742,Z 682.464,A -85,B 0,C 180,E1 -27089.998,E2 -27089.998} C_VEL
LIN {X 0,Y 91.421,Z 680.986,A -85,B 0,C 180,E1 -27094.407,E2 -27094.407} C_VEL
LIN {X 0,Y 91.76,Z 676.983,A -85,B 0,C 180,E1 -27103.282,E2 -27103.282} C_VEL
LIN {X 0,Y 93.839,Z 671.506,A -85,B 0,C 180,E1 -27111.99,E2 -27111.99} C_VEL
LIN {X 0,Y 97.786,Z 664.42,A -85,B 0,C 180,E1 -27120.203,E2 -27120.203} C_VEL
LIN {X 0,Y 102.636,Z 656.761,A -85,B 0,C 180,E1 -27126.807,E2 -27126.807} C_VEL
LIN {X 0,Y 107.743,Z 648.816,A -85,B 0,C 180,E1 -27132.004,E2 -27132.004} C_VEL
LIN {X 0,Y 109.57,Z 645.076,A -85,B 0,C 180,E1 -27134.216,E2 -27134.216} C_VEL
LIN {X 0,Y 111.209,Z 638.575,A -85,B 0,C 180,E1 -27138.012,E2 -27138.012} C_VEL
LIN {X 0,Y 113.104,Z 631.716,A -85,B 0,C 180,E1 -27141.547,E2 -27141.547} C_VEL
LIN {X 0,Y 115.21,Z 627.33,A -85,B 0,C 180,E1 -27143.246,E2 -27143.246} C_VEL
LIN {X 0,Y 122.035,Z 615.345,A -85,B 0,C 180,E1 -27146.619,E2 -27146.619} C_VEL
LIN {X 0,Y 128.649,Z 602.194,A -85,B 0,C 180,E1 -27149.36,E2 -27149.36} C_VEL
LIN {X 0,Y 134.085,Z 589.423,A -85,B 0,C 180,E1 -27151.392,E2 -27151.392} C_VEL
LIN {X 0,Y 139.126,Z 575.534,A -85,B 0,C 180,E1 -27153.023,E2 -27153.023} C_VEL
LIN {X 0,Y 143.301,Z 560.935,A -85,B 0,C 180,E1 -27154.31,E2 -27154.31} C_VEL
LIN {X 0,Y 146.407,Z 546.901,A -85,B 0,C 180,E1 -27155.167,E2 -27155.167} C_VEL
LIN {X 0,Y 148.879,Z 529.479,A -85,B 0,C 180,E1 -27155.923,E2 -27155.923} C_VEL
LIN {X 0,Y 153.722,Z 487.088,A -85,B 0,C 180,E1 -27157.491,E2 -27157.491} C_VEL
LIN {X 0,Y 149.592,Z 474.582,A -85,B 0,C 180,E1 -27160.973,E2 -27160.973} C_VEL
LIN {X 0,Y 146.189,Z 465.287,A -85,B 0,C 180,E1 -27164.088,E2 -27164.088} C_VEL
LIN {X 0,Y 144.021,Z 460.057,A -85,B 0,C 180,E1 -27166.183,E2 -27166.183} C_VEL
LIN {X 0,Y 139.143,Z 451.089,A -85,B 0,C 180,E1 -27171.286,E2 -27171.286} C_VEL
LIN {X 0,Y 134.855,Z 443.596,A -85,B 0,C 180,E1 -27176.906,E2 -27176.906} C_VEL
LIN {X 0,Y 132.857,Z 440.388,A -85,B 0,C 180,E1 -27180.001,E2 -27180.001} C_VEL
LIN {X 0,Y 130.753,Z 436.701,A -85,B 0,C 180,E1 -27184.218,E2 -27184.218} C_VEL
LIN {X 0,Y 128.189,Z 433.154,A -85,B 0,C 180,E1 -27191.328,E2 -27191.328} C_VEL
LIN {X 0,Y 127.835,Z 431.952,A -85,B 0,C 180,E1 -27193.354,E2 -27193.354} C_VEL
LIN {X 0,Y 127.051,Z 431.81,A -85,B 0,C 180,E1 -27202.783,E2 -27202.783} C_VEL
LIN {X 0,Y 127.644,Z 432.204,A -85,B 0,C 180,E1 -27207.27,E2 -27207.27} C_VEL
LIN {X 0,Y 128.848,Z 435.308,A -85,B 0,C 180,E1 -27212.648,E2 -27212.648} C_VEL
LIN {X 0,Y 130.417,Z 437.106,A -85,B 0,C 180,E1 -27216.476,E2 -27216.476} C_VEL
LIN {X 0,Y 133.285,Z 441.769,A -85,B 0,C 180,E1 -27222.021,E2 -27222.021} C_VEL
LIN {X 0,Y 136.009,Z 446.102,A -85,B 0,C 180,E1 -27226.008,E2 -27226.008} C_VEL
LIN {X 0,Y 139.08,Z 451.197,A -85,B 0,C 180,E1 -27229.835,E2 -27229.835} C_VEL
LIN {X 0,Y 143.225,Z 458.602,A -85,B 0,C 180,E1 -27234.192,E2 -27234.192} C_VEL
LIN {X 0,Y 147.675,Z 467.09,A -85,B 0,C 180,E1 -27238.21,E2 -27238.21} C_VEL
LIN {X 0,Y 152.902,Z 477.794,A -85,B 0,C 180,E1 -27242.335,E2 -27242.335} C_VEL
LIN {X 0,Y 153.861,Z 480.168,A -85,B 0,C 180,E1 -27243.065,E2 -27243.065} C_VEL
LIN {X 0,Y 147.835,Z 531.214,A -85,B 0,C 180,E1 -27245.003,E2 -27245.003} C_VEL
LIN {X 0,Y 144.913,Z 546.661,A -85,B 0,C 180,E1 -27245.943,E2 -27245.943} C_VEL
LIN {X 0,Y 141.12,Z 561.674,A -85,B 0,C 180,E1 -27247.298,E2 -27247.298} C_VEL
LIN {X 0,Y 136.584,Z 575.417,A -85,B 0,C 180,E1 -27248.89,E2 -27248.89} C_VEL
LIN {X 0,Y 130.762,Z 590.031,A -85,B 0,C 180,E1 -27251.189,E2 -27251.189} C_VEL
LIN {X 0,Y 124.277,Z 603.664,A -85,B 0,C 180,E1 -27254.026,E2 -27254.026} C_VEL
LIN {X 0,Y 117.554,Z 616.065,A -85,B 0,C 180,E1 -27257.485,E2 -27257.485} C_VEL
LIN {X 0,Y 111.817,Z 625.679,A -85,B 0,C 180,E1 -27260.961,E2 -27260.961} C_VEL
LIN {X 0,Y 104.702,Z 636.593,A -85,B 0,C 180,E1 -27266.153,E2 -27266.153} C_VEL
LIN {X 0,Y 98.456,Z 645.707,A -85,B 0,C 180,E1 -27272.026,E2 -27272.026} C_VEL
LIN {X 0,Y 92.607,Z 654.153,A -85,B 0,C 180,E1 -27279.389,E2 -27279.389} C_VEL
LIN {X 0,Y 88.337,Z 660.813,A -85,B 0,C 180,E1 -27287.305,E2 -27287.305} C_VEL
LIN {X 0,Y 85.518,Z 665.86,A -85,B 0,C 180,E1 -27295.308,E2 -27295.308} C_VEL
LIN {X 0,Y 84.001,Z 669.697,A -85,B 0,C 180,E1 -27303.208,E2 -27303.208} C_VEL
LIN {X 0,Y 83.698,Z 672.926,A -85,B 0,C 180,E1 -27312.205,E2 -27312.205} C_VEL
LIN {X 0,Y 84.464,Z 674.602,A -85,B 0,C 180,E1 -27318.495,E2 -27318.495} C_VEL
LIN {X 0,Y 86.102,Z 675.833,A -85,B 0,C 180,E1 -27325.152,E2 -27325.152} C_VEL
LIN {X 0,Y 88.782,Z 676.542,A -85,B 0,C 180,E1 -27331.641,E2 -27331.641} C_VEL
LIN {X 0,Y 92.299,Z 676.716,A -85,B 0,C 180,E1 -27337.62,E2 -27337.62} C_VEL
LIN {X 0,Y 96.574,Z 676.385,A -85,B 0,C 180,E1 -27343.075,E2 -27343.075} C_VEL
LIN {X 0,Y 101.625,Z 675.489,A -85,B 0,C 180,E1 -27348.024,E2 -27348.024} C_VEL
LIN {X 0,Y 107.258,Z 674.085,A -85,B 0,C 180,E1 -27352.468,E2 -27352.468} C_VEL
LIN {X 0,Y 116.652,Z 671.076,A -85,B 0,C 180,E1 -27358.237,E2 -27358.237} C_VEL
LIN {X 0,Y 127.247,Z 666.748,A -85,B 0,C 180,E1 -27363.165,E2 -27363.165} C_VEL
LIN {X 0,Y 138.647,Z 661.056,A -85,B 0,C 180,E1 -27367.281,E2 -27367.281} C_VEL
LIN {X 0,Y 150.583,Z 653.911,A -85,B 0,C 180,E1 -27370.759,E2 -27370.759} C_VEL
LIN {X 0,Y 162.702,Z 645.258,A -85,B 0,C 180,E1 -27373.616,E2 -27373.616} C_VEL
LIN {X 0,Y 174.477,Z 635.374,A -85,B 0,C 180,E1 -27375.938,E2 -27375.938} C_VEL
LIN {X 0,Y 185.024,Z 624.956,A -85,B 0,C 180,E1 -27377.69,E2 -27377.69} C_VEL
LIN {X 0,Y 193.136,Z 615.61,A -85,B 0,C 180,E1 -27378.893,E2 -27378.893} C_VEL
LIN {X 0,Y 193.268,Z 615.46,A -85,B 0,C 180,E1 -27379.007,E2 -27379.007} C_VEL
LIN {X 0,Y 183.489,Z 626.918,A -85,B 0,C 180,E1 -27380.213,E2 -27380.213} C_VEL
LIN {X 0,Y 172.277,Z 638.152,A -85,B 0,C 180,E1 -27381.86,E2 -27381.86} C_VEL
LIN {X 0,Y 161.218,Z 647.669,A -85,B 0,C 180,E1 -27383.727,E2 -27383.727} C_VEL
LIN {X 0,Y 152.029,Z 654.625,A -85,B 0,C 180,E1 -27385.648,E2 -27385.648} C_VEL
LIN {X 0,Y 140.196,Z 662.526,A -85,B 0,C 180,E1 -27388.683,E2 -27388.683} C_VEL
LIN {X 0,Y 128.874,Z 669.028,A -85,B 0,C 180,E1 -27392.296,E2 -27392.296} C_VEL
LIN {X 0,Y 119.174,Z 673.933,A -85,B 0,C 180,E1 -27396.306,E2 -27396.306} C_VEL
LIN {X 0,Y 111.025,Z 677.471,A -85,B 0,C 180,E1 -27400.567,E2 -27400.567} C_VEL
LIN {X 0,Y 102.172,Z 680.796,A -85,B 0,C 180,E1 -27406.537,E2 -27406.537} C_VEL
LIN {X 0,Y 94.845,Z 683.03,A -85,B 0,C 180,E1 -27413.642,E2 -27413.642} C_VEL
LIN {X 0,Y 89.195,Z 684.249,A -85,B 0,C 180,E1 -27421.784,E2 -27421.784} C_VEL
LIN {X 0,Y 85.589,Z 684.49,A -85,B 0,C 180,E1 -27430.823,E2 -27430.823} C_VEL
LIN {X 0,Y 84.218,Z 683.657,A -85,B 0,C 180,E1 -27440.39,E2 -27440.39} C_VEL
LIN {X 0,Y 84.461,Z 682.523,A -85,B 0,C 180,E1 -27446.852,E2 -27446.852} C_VEL
LIN {X 0,Y 84.68,Z 681.71,A -85,B 0,C 180,E1 -27449.998,E2 -27449.998} C_VEL
LIN {X 0,Y 84.329,Z 680.146,A -85,B 0,C 180,E1 -27454.778,E2 -27454.778} C_VEL
LIN {X 0,Y 84.817,Z 675.97,A -85,B 0,C 180,E1 -27464.391,E2 -27464.391} C_VEL
LIN {X 0,Y 87.236,Z 670.311,A -85,B 0,C 180,E1 -27473.752,E2 -27473.752} C_VEL
LIN {X 0,Y 91.716,Z 662.936,A -85,B 0,C 180,E1 -27482.554,E2 -27482.554} C_VEL
LIN {X 0,Y 96.985,Z 655.163,A -85,B 0,C 180,E1 -27489.348,E2 -27489.348} C_VEL
LIN {X 0,Y 102.458,Z 647.131,A -85,B 0,C 180,E1 -27494.673,E2 -27494.673} C_VEL
LIN {X 0,Y 109.892,Z 635.897,A -85,B 0,C 180,E1 -27500.122,E2 -27500.122} C_VEL
LIN {X 0,Y 115.21,Z 627.33,A -85,B 0,C 180,E1 -27503.246,E2 -27503.246} C_VEL
LIN {X 0,Y 117.332,Z 622.86,A -85,B 0,C 180,E1 -27504.842,E2 -27504.842} C_VEL
LIN {X 0,Y 119.413,Z 615.26,A -85,B 0,C 180,E1 -27507.767,E2 -27507.767} C_VEL
LIN {X 0,Y 121.492,Z 607.37,A -85,B 0,C 180,E1 -27510.441,E2 -27510.441} C_VEL
LIN {X 0,Y 123.517,Z 602.363,A -85,B 0,C 180,E1 -27511.602,E2 -27511.602} C_VEL
LIN {X 0,Y 129.356,Z 589.168,A -85,B 0,C 180,E1 -27513.693,E2 -27513.693} C_VEL
LIN {X 0,Y 134.692,Z 574.908,A -85,B 0,C 180,E1 -27515.329,E2 -27515.329} C_VEL
LIN {X 0,Y 139.038,Z 560.073,A -85,B 0,C 180,E1 -27516.595,E2 -27516.595} C_VEL
LIN {X 0,Y 142.221,Z 545.826,A -85,B 0,C 180,E1 -27517.434,E2 -27517.434} C_VEL
LIN {X 0,Y 144.996,Z 526.025,A -85,B 0,C 180,E1 -27518.259,E2 -27518.259} C_VEL
LIN {X 0,Y 149.332,Z 489.427,A -85,B 0,C 180,E1 -27519.584,E2 -27519.584} C_VEL
LIN {X 0,Y 145.352,Z 476.864,A -85,B 0,C 180,E1 -27523.317,E2 -27523.317} C_VEL
LIN {X 0,Y 141.681,Z 466.541,A -85,B 0,C 180,E1 -27527.088,E2 -27527.088} C_VEL
LIN {X 0,Y 136.884,Z 457.26,A -85,B 0,C 180,E1 -27532.407,E2 -27532.407} C_VEL
LIN {X 0,Y 132.85,Z 449.822,A -85,B 0,C 180,E1 -27538.078,E2 -27538.078} C_VEL
LIN {X 0,Y 131.033,Z 446.799,A -85,B 0,C 180,E1 -27541.148,E2 -27541.148} C_VEL
LIN {X 0,Y 128.901,Z 442.953,A -85,B 0,C 180,E1 -27545.838,E2 -27545.838} C_VEL
LIN {X 0,Y 126.99,Z 440.112,A -85,B 0,C 180,E1 -27551.802,E2 -27551.802} C_VEL
LIN {X 0,Y 126.717,Z 439.057,A -85,B 0,C 180,E1 -27553.474,E2 -27553.474} C_VEL
LIN {X 0,Y 125.941,Z 438.717,A -85,B 0,C 180,E1 -27559.563,E2 -27559.563} C_VEL
LIN {X 0,Y 126.453,Z 439.088,A -85,B 0,C 180,E1 -27566.63,E2 -27566.63} C_VEL
LIN {X 0,Y 127.717,Z 442.422,A -85,B 0,C 180,E1 -27572.561,E2 -27572.561} C_VEL
LIN {X 0,Y 128.971,Z 443.937,A -85,B 0,C 180,E1 -27575.781,E2 -27575.781} C_VEL
LIN {X 0,Y 131.695,Z 448.592,A -85,B 0,C 180,E1 -27581.347,E2 -27581.347} C_VEL
LIN {X 0,Y 134.317,Z 452.952,A -85,B 0,C 180,E1 -27585.36,E2 -27585.36} C_VEL
LIN {X 0,Y 137.258,Z 458.15,A -85,B 0,C 180,E1 -27589.231,E2 -27589.231} C_VEL
LIN {X 0,Y 140.957,Z 465.176,A -85,B 0,C 180,E1 -27593.307,E2 -27593.307} C_VEL
LIN {X 0,Y 144.703,Z 472.774,A -85,B 0,C 180,E1 -27596.952,E2 -27596.952} C_VEL
LIN {X 0,Y 149.326,Z 482.468,A -85,B 0,C 180,E1 -27600.827,E2 -27600.827} C_VEL
LIN {X 0,Y 149.488,Z 482.879,A -85,B 0,C 180,E1 -27600.962,E2 -27600.962} C_VEL
LIN {X 0,Y 143.651,Z 530.969,A -85,B 0,C 180,E1 -27602.754,E2 -27602.754} C_VEL
LIN {X 0,Y 140.631,Z 546.6,A -85,B 0,C 180,E1 -27603.672,E2 -27603.672} C_VEL
LIN {X 0,Y 136.519,Z 562.323,A -85,B 0,C 180,E1 -27605.073,E2 -27605.073} C_VEL
LIN {X 0,Y 131.489,Z 576.953,A -85,B 0,C 180,E1 -27606.786,E2 -27606.786} C_VEL
LIN {X 0,Y 125.465,Z 591.368,A -85,B 0,C 180,E1 -27609.079,E2 -27609.079} C_VEL
LIN {X 0,Y 118.778,Z 604.766,A -85,B 0,C 180,E1 -27611.904,E2 -27611.904} C_VEL
LIN {X 0,Y 111.692,Z 617.141,A -85,B 0,C 180,E1 -27615.424,E2 -27615.424} C_VEL
LIN {X 0,Y 105.045,Z 627.615,A -85,B 0,C 180,E1 -27619.4,E2 -27619.4} C_VEL
LIN {X 0,Y 97.899,Z 637.959,A -85,B 0,C 180,E1 -27624.669,E2 -27624.669} C_VEL
LIN {X 0,Y 91.377,Z 646.916,A -85,B 0,C 180,E1 -27630.874,E2 -27630.874} C_VEL
LIN {X 0,Y 85.336,Z 655.188,A -85,B 0,C 180,E1 -27638.767,E2 -27638.767} C_VEL
LIN {X 0,Y 80.976,Z 661.72,A -85,B 0,C 180,E1 -27647.304,E2 -27647.304} C_VEL
LIN {X 0,Y 77.973,Z 667.053,A -85,B 0,C 180,E1 -27656.789,E2 -27656.789} C_VEL
LIN {X 0,Y 76.75,Z 670.334,A -85,B 0,C 180,E1 -27664.496,E2 -27664.496} C_VEL
LIN {X 0,Y 76.635,Z 673.078,A -85,B 0,C 180,E1 -27672.803,E2 -27672.803} C_VEL
LIN {X 0,Y 78.454,Z 675.612,A -85,B 0,C 180,E1 -27683.733,E2 -27683.733} C_VEL
LIN {X 0,Y 83.025,Z 677.012,A -85,B 0,C 180,E1 -27694.958,E2 -27694.958} C_VEL
LIN {X 0,Y 88.308,Z 677.143,A -85,B 0,C 180,E1 -27702.757,E2 -27702.757} C_VEL
LIN {X 0,Y 97.465,Z 675.944,A -85,B 0,C 180,E1 -27711.707,E2 -27711.707} C_VEL
LIN {X 0,Y 105.54,Z 674.048,A -85,B 0,C 180,E1 -27717.3,E2 -27717.3} C_VEL
LIN {X 0,Y 112.472,Z 671.973,A -85,B 0,C 180,E1 -27721.101,E2 -27721.101} C_VEL
LIN {X 0,Y 125.037,Z 667.186,A -85,B 0,C 180,E1 -27726.453,E2 -27726.453} C_VEL
LIN {X 0,Y 135.56,Z 662.217,A -85,B 0,C 180,E1 -27729.917,E2 -27729.917} C_VEL
LIN {X 0,Y 146.635,Z 656.004,A -85,B 0,C 180,E1 -27732.922,E2 -27732.922} C_VEL
LIN {X 0,Y 158.091,Z 648.506,A -85,B 0,C 180,E1 -27735.469,E2 -27735.469} C_VEL
LIN {X 0,Y 169.597,Z 639.636,A -85,B 0,C 180,E1 -27737.613,E2 -27737.613} C_VEL
LIN {X 0,Y 175.882,Z 634.126,A -85,B 0,C 180,E1 -27738.642,E2 -27738.642} C_VEL
LIN {X 0,Y 174.082,Z 635.867,A -85,B 0,C 180,E1 -27739.079,E2 -27739.079} C_VEL
LIN {X 0,Y 161.747,Z 646.457,A -85,B 0,C 180,E1 -27740.9,E2 -27740.9} C_VEL
LIN {X 0,Y 150.647,Z 654.582,A -85,B 0,C 180,E1 -27742.869,E2 -27742.869} C_VEL
LIN {X 0,Y 140.01,Z 661.452,A -85,B 0,C 180,E1 -27745.371,E2 -27745.371} C_VEL
LIN {X 0,Y 128.111,Z 668.081,A -85,B 0,C 180,E1 -27748.626,E2 -27748.626} C_VEL
LIN {X 0,Y 116.108,Z 673.762,A -85,B 0,C 180,E1 -27753.007,E2 -27753.007} C_VEL
LIN {X 0,Y 106.508,Z 677.587,A -85,B 0,C 180,E1 -27757.641,E2 -27757.641} C_VEL
LIN {X 0,Y 97.09,Z 680.704,A -85,B 0,C 180,E1 -27763.623,E2 -27763.623} C_VEL
LIN {X 0,Y 89.165,Z 682.825,A -85,B 0,C 180,E1 -27770.906,E2 -27770.906} C_VEL
LIN {X 0,Y 82.949,Z 683.874,A -85,B 0,C 180,E1 -27779.443,E2 -27779.443} C_VEL
LIN {X 0,Y 78.857,Z 683.944,A -85,B 0,C 180,E1 -27789.113,E2 -27789.113} C_VEL
LIN {X 0,Y 77.195,Z 683.019,A -85,B 0,C 180,E1 -27799.506,E2 -27799.506} C_VEL
LIN {X 0,Y 77.414,Z 681.657,A -85,B 0,C 180,E1 -27806.974,E2 -27806.974} C_VEL
LIN {X 0,Y 77.616,Z 680.925,A -85,B 0,C 180,E1 -27809.998,E2 -27809.998} C_VEL
LIN {X 0,Y 77.332,Z 677.284,A -85,B 0,C 180,E1 -27820.47,E2 -27820.47} C_VEL
LIN {X 0,Y 79.023,Z 672.206,A -85,B 0,C 180,E1 -27830.837,E2 -27830.837} C_VEL
LIN {X 0,Y 82.923,Z 665.575,A -85,B 0,C 180,E1 -27840.563,E2 -27840.563} C_VEL
LIN {X 0,Y 88.009,Z 658.353,A -85,B 0,C 180,E1 -27848.232,E2 -27848.232} C_VEL
LIN {X 0,Y 94.378,Z 649.578,A -85,B 0,C 180,E1 -27855.023,E2 -27855.023} C_VEL
LIN {X 0,Y 101.843,Z 639.047,A -85,B 0,C 180,E1 -27860.85,E2 -27860.85} C_VEL
LIN {X 0,Y 109.677,Z 627.194,A -85,B 0,C 180,E1 -27865.506,E2 -27865.506} C_VEL
LIN {X 0,Y 116.893,Z 615.05,A -85,B 0,C 180,E1 -27868.952,E2 -27868.952} C_VEL
LIN {X 0,Y 123.517,Z 602.363,A -85,B 0,C 180,E1 -27871.602,E2 -27871.602} C_VEL
LIN {X 0,Y 125.463,Z 597.329,A -85,B 0,C 180,E1 -27872.685,E2 -27872.685} C_VEL
LIN {X 0,Y 127.229,Z 588.86,A -85,B 0,C 180,E1 -27874.904,E2 -27874.904} C_VEL
LIN {X 0,Y 128.782,Z 580.211,A -85,B 0,C 180,E1 -27876.947,E2 -27876.947} C_VEL
LIN {X 0,Y 130.309,Z 574.741,A -85,B 0,C 180,E1 -27877.734,E2 -27877.734} C_VEL
LIN {X 0,Y 134.641,Z 560.499,A -85,B 0,C 180,E1 -27878.934,E2 -27878.934} C_VEL
LIN {X 0,Y 138.081,Z 545.721,A -85,B 0,C 180,E1 -27879.785,E2 -27879.785} C_VEL
LIN {X 0,Y 140.897,Z 526.532,A -85,B 0,C 180,E1 -27880.567,E2 -27880.567} C_VEL
LIN {X 0,Y 145.123,Z 491.779,A -85,B 0,C 180,E1 -27881.813,E2 -27881.813} C_VEL
LIN {X 0,Y 141.235,Z 479.041,A -85,B 0,C 180,E1 -27885.834,E2 -27885.834} C_VEL
LIN {X 0,Y 138.538,Z 471.238,A -85,B 0,C 180,E1 -27888.957,E2 -27888.957} C_VEL
LIN {X 0,Y 134.356,Z 462.833,A -85,B 0,C 180,E1 -27893.996,E2 -27893.996} C_VEL
LIN {X 0,Y 130.716,Z 455.812,A -85,B 0,C 180,E1 -27899.58,E2 -27899.58} C_VEL
LIN {X 0,Y 129.388,Z 453.373,A -85,B 0,C 180,E1 -27902.086,E2 -27902.086} C_VEL
LIN {X 0,Y 127.581,Z 449.847,A -85,B 0,C 180,E1 -27906.326,E2 -27906.326} C_VEL
LIN {X 0,Y 125.766,Z 446.931,A -85,B 0,C 180,E1 -27912.51,E2 -27912.51} C_VEL
LIN {X 0,Y 125.476,Z 445.934,A -85,B 0,C 180,E1 -27914.273,E2 -27914.273} C_VEL
LIN {X 0,Y 124.946,Z 445.842,A -85,B 0,C 180,E1 -27923.189,E2 -27923.189} C_VEL
LIN {X 0,Y 125.325,Z 446.242,A -85,B 0,C 180,E1 -27926.443,E2 -27926.443} C_VEL
LIN {X 0,Y 126.474,Z 449.342,A -85,B 0,C 180,E1 -27932.1,E2 -27932.1} C_VEL
LIN {X 0,Y 127.541,Z 450.736,A -85,B 0,C 180,E1 -27935.054,E2 -27935.054} C_VEL
LIN {X 0,Y 130.06,Z 455.279,A -85,B 0,C 180,E1 -27940.537,E2 -27940.537} C_VEL
LIN {X 0,Y 132.435,Z 459.522,A -85,B 0,C 180,E1 -27944.452,E2 -27944.452} C_VEL
LIN {X 0,Y 134.922,Z 464.099,A -85,B 0,C 180,E1 -27947.931,E2 -27947.931} C_VEL
LIN {X 0,Y 138.554,Z 471.405,A -85,B 0,C 180,E1 -27952.249,E2 -27952.249} C_VEL
LIN {X 0,Y 142.023,Z 478.855,A -85,B 0,C 180,E1 -27955.847,E2 -27955.847} C_VEL
LIN {X 0,Y 145.255,Z 485.887,A -85,B 0,C 180,E1 -27958.783,E2 -27958.783} C_VEL
LIN {X 0,Y 139.411,Z 531.833,A -85,B 0,C 180,E1 -27960.438,E2 -27960.438} C_VEL
LIN {X 0,Y 136.268,Z 547.54,A -85,B 0,C 180,E1 -27961.37,E2 -27961.37} C_VEL
LIN {X 0,Y 132.154,Z 562.703,A -85,B 0,C 180,E1 -27962.7,E2 -27962.7} C_VEL
LIN {X 0,Y 127.388,Z 576.218,A -85,B 0,C 180,E1 -27964.217,E2 -27964.217} C_VEL
LIN {X 0,Y 121.072,Z 590.947,A -85,B 0,C 180,E1 -27966.481,E2 -27966.481} C_VEL
LIN {X 0,Y 114.434,Z 603.922,A -85,B 0,C 180,E1 -27969.132,E2 -27969.132} C_VEL
LIN {X 0,Y 107.507,Z 615.799,A -85,B 0,C 180,E1 -27972.403,E2 -27972.403} C_VEL
LIN {X 0,Y 100.146,Z 626.975,A -85,B 0,C 180,E1 -27976.522,E2 -27976.522} C_VEL
LIN {X 0,Y 92.247,Z 637.862,A -85,B 0,C 180,E1 -27982.077,E2 -27982.077} C_VEL
LIN {X 0,Y 85.189,Z 647.034,A -85,B 0,C 180,E1 -27988.614,E2 -27988.614} C_VEL
LIN {X 0,Y 79.037,Z 654.974,A -85,B 0,C 180,E1 -27996.498,E2 -27996.498} C_VEL
LIN {X 0,Y 73.842,Z 662.192,A -85,B 0,C 180,E1 -28006.593,E2 -28006.593} C_VEL
LIN {X 0,Y 70.807,Z 667.377,A -85,B 0,C 180,E1 -28016.704,E2 -28016.704} C_VEL
LIN {X 0,Y 69.441,Z 671.391,A -85,B 0,C 180,E1 -28027.394,E2 -28027.394} C_VEL
LIN {X 0,Y 69.703,Z 673.628,A -85,B 0,C 180,E1 -28035.103,E2 -28035.103} C_VEL
LIN {X 0,Y 71.198,Z 675.564,A -85,B 0,C 180,E1 -28043.68,E2 -28043.68} C_VEL
LIN {X 0,Y 73.794,Z 676.798,A -85,B 0,C 180,E1 -28051.561,E2 -28051.561} C_VEL
LIN {X 0,Y 77.557,Z 677.484,A -85,B 0,C 180,E1 -28058.746,E2 -28058.746} C_VEL
LIN {X 0,Y 85.876,Z 677.434,A -85,B 0,C 180,E1 -28069.143,E2 -28069.143} C_VEL
LIN {X 0,Y 93.755,Z 676.407,A -85,B 0,C 180,E1 -28075.699,E2 -28075.699} C_VEL
LIN {X 0,Y 100.474,Z 675.001,A -85,B 0,C 180,E1 -28079.999,E2 -28079.999} C_VEL
LIN {X 0,Y 107.635,Z 673.108,A -85,B 0,C 180,E1 -28083.742,E2 -28083.742} C_VEL
LIN {X 0,Y 117.82,Z 669.748,A -85,B 0,C 180,E1 -28087.977,E2 -28087.977} C_VEL
LIN {X 0,Y 129.174,Z 665.101,A -85,B 0,C 180,E1 -28091.662,E2 -28091.662} C_VEL
LIN {X 0,Y 142.695,Z 658.294,A -85,B 0,C 180,E1 -28095.152,E2 -28095.152} C_VEL
LIN {X 0,Y 154.897,Z 650.853,A -85,B 0,C 180,E1 -28097.668,E2 -28097.668} C_VEL
LIN {X 0,Y 157.708,Z 648.896,A -85,B 0,C 180,E1 -28098.175,E2 -28098.175} C_VEL
LIN {X 0,Y 156.117,Z 650.131,A -85,B 0,C 180,E1 -28099.024,E2 -28099.024} C_VEL
LIN {X 0,Y 146.497,Z 656.63,A -85,B 0,C 180,E1 -28100.69,E2 -28100.69} C_VEL
LIN {X 0,Y 134.006,Z 663.972,A -85,B 0,C 180,E1 -28103.391,E2 -28103.391} C_VEL
LIN {X 0,Y 121.884,Z 669.998,A -85,B 0,C 180,E1 -28106.648,E2 -28106.648} C_VEL
LIN {X 0,Y 107.647,Z 675.855,A -85,B 0,C 180,E1 -28111.923,E2 -28111.923} C_VEL
LIN {X 0,Y 97.151,Z 679.293,A -85,B 0,C 180,E1 -28117.271,E2 -28117.271} C_VEL
LIN {X 0,Y 87.818,Z 681.706,A -85,B 0,C 180,E1 -28123.921,E2 -28123.921} C_VEL
LIN {X 0,Y 79.744,Z 683.186,A -85,B 0,C 180,E1 -28132.482,E2 -28132.482} C_VEL
LIN {X 0,Y 74.243,Z 683.568,A -85,B 0,C 180,E1 -28141.748,E2 -28141.748} C_VEL
LIN {X 0,Y 70.878,Z 682.973,A -85,B 0,C 180,E1 -28152.692,E2 -28152.692} C_VEL
LIN {X 0,Y 70.158,Z 681.377,A -85,B 0,C 180,E1 -28164.248,E2 -28164.248} C_VEL
LIN {X 0,Y 70.534,Z 680.133,A -85,B 0,C 180,E1 -28169.997,E2 -28169.997} C_VEL
LIN {X 0,Y 70.338,Z 676.319,A -85,B 0,C 180,E1 -28181.525,E2 -28181.525} C_VEL
LIN {X 0,Y 72.371,Z 671.047,A -85,B 0,C 180,E1 -28192.855,E2 -28192.855} C_VEL
LIN {X 0,Y 76.834,Z 664.214,A -85,B 0,C 180,E1 -28203.283,E2 -28203.283} C_VEL
LIN {X 0,Y 82.485,Z 656.769,A -85,B 0,C 180,E1 -28211.322,E2 -28211.322} C_VEL
LIN {X 0,Y 89.433,Z 647.753,A -85,B 0,C 180,E1 -28218.289,E2 -28218.289} C_VEL
LIN {X 0,Y 96.296,Z 638.538,A -85,B 0,C 180,E1 -28223.396,E2 -28223.396} C_VEL
LIN {X 0,Y 103.864,Z 627.676,A -85,B 0,C 180,E1 -28227.756,E2 -28227.756} C_VEL
LIN {X 0,Y 111.265,Z 615.839,A -85,B 0,C 180,E1 -28231.208,E2 -28231.208} C_VEL
LIN {X 0,Y 118.323,Z 602.967,A -85,B 0,C 180,E1 -28233.941,E2 -28233.941} C_VEL
LIN {X 0,Y 124.122,Z 590.582,A -85,B 0,C 180,E1 -28235.923,E2 -28235.923} C_VEL
LIN {X 0,Y 129.769,Z 576.216,A -85,B 0,C 180,E1 -28237.61,E2 -28237.61} C_VEL
LIN {X 0,Y 130.309,Z 574.741,A -85,B 0,C 180,E1 -28237.734,E2 -28237.734} C_VEL
LIN {X 0,Y 131.734,Z 569.297,A -85,B 0,C 180,E1 -28238.457,E2 -28238.457} C_VEL
LIN {X 0,Y 132.739,Z 560.187,A -85,B 0,C 180,E1 -28240.142,E2 -28240.142} C_VEL
LIN {X 0,Y 133.37,Z 550.969,A -85,B 0,C 180,E1 -28241.726,E2 -28241.726} C_VEL
LIN {X 0,Y 134.142,Z 545.23,A -85,B 0,C 180,E1 -28242.273,E2 -28242.273} C_VEL
LIN {X 0,Y 137.044,Z 526.046,A -85,B 0,C 180,E1 -28243.017,E2 -28243.017} C_VEL
LIN {X 0,Y 141.027,Z 494.119,A -85,B 0,C 180,E1 -28244.14,E2 -28244.14} C_VEL
LIN {X 0,Y 137.558,Z 481.978,A -85,B 0,C 180,E1 -28248.267,E2 -28248.267} C_VEL
LIN {X 0,Y 135.563,Z 476.168,A -85,B 0,C 180,E1 -28250.75,E2 -28250.75} C_VEL
LIN {X 0,Y 131.9,Z 468.326,A -85,B 0,C 180,E1 -28255.7,E2 -28255.7} C_VEL
LIN {X 0,Y 128.832,Z 462.041,A -85,B 0,C 180,E1 -28260.843,E2 -28260.843} C_VEL
LIN {X 0,Y 127.588,Z 459.583,A -85,B 0,C 180,E1 -28263.48,E2 -28263.48} C_VEL
LIN {X 0,Y 126.091,Z 456.551,A -85,B 0,C 180,E1 -28267.281,E2 -28267.281} C_VEL
LIN {X 0,Y 124.523,Z 453.706,A -85,B 0,C 180,E1 -28273.299,E2 -28273.299} C_VEL
LIN {X 0,Y 124.363,Z 453.039,A -85,B 0,C 180,E1 -28274.404,E2 -28274.404} C_VEL
LIN {X 0,Y 123.894,Z 452.871,A -85,B 0,C 180,E1 -28283.397,E2 -28283.397} C_VEL
LIN {X 0,Y 124.173,Z 453.25,A -85,B 0,C 180,E1 -28286.001,E2 -28286.001} C_VEL
LIN {X 0,Y 125.35,Z 456.413,A -85,B 0,C 180,E1 -28292.002,E2 -28292.002} C_VEL
LIN {X 0,Y 126.195,Z 457.696,A -85,B 0,C 180,E1 -28294.503,E2 -28294.503} C_VEL
LIN {X 0,Y 128.299,Z 461.662,A -85,B 0,C 180,E1 -28299.391,E2 -28299.391} C_VEL
LIN {X 0,Y 130.863,Z 466.516,A -85,B 0,C 180,E1 -28303.938,E2 -28303.938} C_VEL
LIN {X 0,Y 133.618,Z 472.116,A -85,B 0,C 180,E1 -28307.943,E2 -28307.943} C_VEL
LIN {X 0,Y 137.655,Z 480.812,A -85,B 0,C 180,E1 -28312.81,E2 -28312.81} C_VEL
LIN {X 0,Y 141.163,Z 488.981,A -85,B 0,C 180,E1 -28316.475,E2 -28316.475} C_VEL
LIN {X 0,Y 135.417,Z 532.574,A -85,B 0,C 180,E1 -28318.003,E2 -28318.003} C_VEL
LIN {X 0,Y 132.284,Z 547.757,A -85,B 0,C 180,E1 -28318.872,E2 -28318.872} C_VEL
LIN {X 0,Y 128.07,Z 562.86,A -85,B 0,C 180,E1 -28320.152,E2 -28320.152} C_VEL
LIN {X 0,Y 122.614,Z 577.684,A -85,B 0,C 180,E1 -28321.781,E2 -28321.781} C_VEL
LIN {X 0,Y 116.516,Z 591.396,A -85,B 0,C 180,E1 -28323.864,E2 -28323.864} C_VEL
LIN {X 0,Y 109.758,Z 604.145,A -85,B 0,C 180,E1 -28326.411,E2 -28326.411} C_VEL
LIN {X 0,Y 102.046,Z 616.744,A -85,B 0,C 180,E1 -28329.86,E2 -28329.86} C_VEL
LIN {X 0,Y 94.465,Z 627.703,A -85,B 0,C 180,E1 -28333.959,E2 -28333.959} C_VEL
LIN {X 0,Y 86.655,Z 637.953,A -85,B 0,C 180,E1 -28339.277,E2 -28339.277} C_VEL
LIN {X 0,Y 78.778,Z 647.607,A -85,B 0,C 180,E1 -28346.453,E2 -28346.453} C_VEL
LIN {X 0,Y 72.654,Z 654.949,A -85,B 0,C 180,E1 -28354.163,E2 -28354.163} C_VEL
LIN {X 0,Y 67.248,Z 661.898,A -85,B 0,C 180,E1 -28364.467,E2 -28364.467} C_VEL
LIN {X 0,Y 63.727,Z 667.479,A -85,B 0,C 180,E1 -28376.179,E2 -28376.179} C_VEL
LIN {X 0,Y 62.327,Z 671.526,A -85,B 0,C 180,E1 -28387.874,E2 -28387.874} C_VEL
LIN {X 0,Y 63.355,Z 674.841,A -85,B 0,C 180,E1 -28400.947,E2 -28400.947} C_VEL
LIN {X 0,Y 65.469,Z 676.365,A -85,B 0,C 180,E1 -28409.186,E2 -28409.186} C_VEL
LIN {X 0,Y 68.754,Z 677.423,A -85,B 0,C 180,E1 -28416.93,E2 -28416.93} C_VEL
LIN {X 0,Y 73.118,Z 678.011,A -85,B 0,C 180,E1 -28423.992,E2 -28423.992} C_VEL
LIN {X 0,Y 78.432,Z 678.118,A -85,B 0,C 180,E1 -28430.302,E2 -28430.302} C_VEL
LIN {X 0,Y 84.569,Z 677.68,A -85,B 0,C 180,E1 -28435.77,E2 -28435.77} C_VEL
LIN {X 0,Y 91.371,Z 676.737,A -85,B 0,C 180,E1 -28440.508,E2 -28440.508} C_VEL
LIN {X 0,Y 98.711,Z 675.288,A -85,B 0,C 180,E1 -28444.587,E2 -28444.587} C_VEL
LIN {X 0,Y 109.971,Z 672.285,A -85,B 0,C 180,E1 -28449.421,E2 -28449.421} C_VEL
LIN {X 0,Y 122.924,Z 667.742,A -85,B 0,C 180,E1 -28453.596,E2 -28453.596} C_VEL
LIN {X 0,Y 137.427,Z 661.217,A -85,B 0,C 180,E1 -28457.186,E2 -28457.186} C_VEL
LIN {X 0,Y 141.048,Z 659.374,A -85,B 0,C 180,E1 -28457.948,E2 -28457.948} C_VEL
LIN {X 0,Y 140.965,Z 659.497,A -85,B 0,C 180,E1 -28458.685,E2 -28458.685} C_VEL
LIN {X 0,Y 128.198,Z 666.243,A -85,B 0,C 180,E1 -28461.253,E2 -28461.253} C_VEL
LIN {X 0,Y 115.822,Z 671.683,A -85,B 0,C 180,E1 -28464.465,E2 -28464.465} C_VEL
LIN {X 0,Y 104.047,Z 676.01,A -85,B 0,C 180,E1 -28468.582,E2 -28468.582} C_VEL
LIN {X 0,Y 92.993,Z 679.309,A -85,B 0,C 180,E1 -28473.761,E2 -28473.761} C_VEL
LIN {X 0,Y 82.995,Z 681.529,A -85,B 0,C 180,E1 -28480.346,E2 -28480.346} C_VEL
LIN {X 0,Y 73.702,Z 682.86,A -85,B 0,C 180,E1 -28489.714,E2 -28489.714} C_VEL
LIN {X 0,Y 68.022,Z 683.092,A -85,B 0,C 180,E1 -28498.893,E2 -28498.893} C_VEL
LIN {X 0,Y 64.102,Z 682.334,A -85,B 0,C 180,E1 -28510.794,E2 -28510.794} C_VEL
LIN {X 0,Y 63.113,Z 680.563,A -85,B 0,C 180,E1 -28523.604,E2 -28523.604} C_VEL
LIN {X 0,Y 63.447,Z 679.248,A -85,B 0,C 180,E1 -28529.997,E2 -28529.997} C_VEL
LIN {X 0,Y 63.362,Z 675.299,A -85,B 0,C 180,E1 -28542.814,E2 -28542.814} C_VEL
LIN {X 0,Y 65.83,Z 669.859,A -85,B 0,C 180,E1 -28555.277,E2 -28555.277} C_VEL
LIN {X 0,Y 70.954,Z 662.807,A -85,B 0,C 180,E1 -28566.46,E2 -28566.46} C_VEL
LIN {X 0,Y 77.222,Z 655.174,A -85,B 0,C 180,E1 -28574.853,E2 -28574.853} C_VEL
LIN {X 0,Y 84.804,Z 645.907,A -85,B 0,C 180,E1 -28581.93,E2 -28581.93} C_VEL
LIN {X 0,Y 93.115,Z 635.225,A -85,B 0,C 180,E1 -28587.519,E2 -28587.519} C_VEL
LIN {X 0,Y 101.597,Z 623.164,A -85,B 0,C 180,E1 -28591.879,E2 -28591.879} C_VEL
LIN {X 0,Y 109.463,Z 610.532,A -85,B 0,C 180,E1 -28595.075,E2 -28595.075} C_VEL
LIN {X 0,Y 116.105,Z 598.146,A -85,B 0,C 180,E1 -28597.38,E2 -28597.38} C_VEL
LIN {X 0,Y 122.152,Z 584.839,A -85,B 0,C 180,E1 -28599.215,E2 -28599.215} C_VEL
LIN {X 0,Y 127.83,Z 569.561,A -85,B 0,C 180,E1 -28600.716,E2 -28600.716} C_VEL
LIN {X 0,Y 132.247,Z 554.096,A -85,B 0,C 180,E1 -28601.786,E2 -28601.786} C_VEL
LIN {X 0,Y 134.142,Z 545.23,A -85,B 0,C 180,E1 -28602.273,E2 -28602.273} C_VEL
LIN {X 0,Y 134.833,Z 539.478,A -85,B 0,C 180,E1 -28602.773,E2 -28602.773} C_VEL
LIN {X 0,Y 134.484,Z 520.698,A -85,B 0,C 180,E1 -28605.479,E2 -28605.479} C_VEL
LIN {X 0,Y 134.856,Z 514.891,A -85,B 0,C 180,E1 -28605.947,E2 -28605.947} C_VEL
LIN {X 0,Y 137.204,Z 496.646,A -85,B 0,C 180,E1 -28606.563,E2 -28606.563} C_VEL
LIN {X 0,Y 134.417,Z 486.363,A -85,B 0,C 180,E1 -28610.246,E2 -28610.246} C_VEL
LIN {X 0,Y 132.843,Z 481.399,A -85,B 0,C 180,E1 -28612.452,E2 -28612.452} C_VEL
LIN {X 0,Y 129.198,Z 473.079,A -85,B 0,C 180,E1 -28617.974,E2 -28617.974} C_VEL
LIN {X 0,Y 126.615,Z 467.321,A -85,B 0,C 180,E1 -28623.06,E2 -28623.06} C_VEL
LIN {X 0,Y 124.644,Z 463.28,A -85,B 0,C 180,E1 -28628.232,E2 -28628.232} C_VEL
LIN {X 0,Y 123.245,Z 460.186,A -85,B 0,C 180,E1 -28634.538,E2 -28634.538} C_VEL
LIN {X 0,Y 122.951,Z 459.828,A -85,B 0,C 180,E1 -28636.608,E2 -28636.608} C_VEL
LIN {X 0,Y 123.01,Z 460.05,A -85,B 0,C 180,E1 -28645.22,E2 -28645.22} C_VEL
LIN {X 0,Y 124.114,Z 463.314,A -85,B 0,C 180,E1 -28651.51,E2 -28651.51} C_VEL
LIN {X 0,Y 124.803,Z 464.505,A -85,B 0,C 180,E1 -28653.756,E2 -28653.756} C_VEL
LIN {X 0,Y 126.751,Z 468.401,A -85,B 0,C 180,E1 -28658.585,E2 -28658.585} C_VEL
LIN {X 0,Y 128.865,Z 472.731,A -85,B 0,C 180,E1 -28662.705,E2 -28662.705} C_VEL
LIN {X 0,Y 131.652,Z 478.69,A -85,B 0,C 180,E1 -28667.023,E2 -28667.023} C_VEL
LIN {X 0,Y 135.354,Z 487.388,A -85,B 0,C 180,E1 -28671.857,E2 -28671.857} C_VEL
LIN {X 0,Y 137.306,Z 492.138,A -85,B 0,C 180,E1 -28674.048,E2 -28674.048} C_VEL
LIN {X 0,Y 131.864,Z 532.343,A -85,B 0,C 180,E1 -28675.38,E2 -28675.38} C_VEL
LIN {X 0,Y 128.61,Z 547.754,A -85,B 0,C 180,E1 -28676.204,E2 -28676.204} C_VEL
LIN {X 0,Y 124.098,Z 563.395,A -85,B 0,C 180,E1 -28677.472,E2 -28677.472} C_VEL
LIN {X 0,Y 118.993,Z 576.988,A -85,B 0,C 180,E1 -28678.884,E2 -28678.884} C_VEL
LIN {X 0,Y 112.597,Z 591.049,A -85,B 0,C 180,E1 -28680.911,E2 -28680.911} C_VEL
LIN {X 0,Y 105.665,Z 603.757,A -85,B 0,C 180,E1 -28683.325,E2 -28683.325} C_VEL
LIN {X 0,Y 97.947,Z 616.002,A -85,B 0,C 180,E1 -28686.535,E2 -28686.535} C_VEL
LIN {X 0,Y 90.318,Z 626.628,A -85,B 0,C 180,E1 -28690.357,E2 -28690.357} C_VEL
LIN {X 0,Y 82.557,Z 636.389,A -85,B 0,C 180,E1 -28695.206,E2 -28695.206} C_VEL
LIN {X 0,Y 74.454,Z 645.816,A -85,B 0,C 180,E1 -28701.863,E2 -28701.863} C_VEL
LIN {X 0,Y 67.358,Z 653.764,A -85,B 0,C 180,E1 -28710.003,E2 -28710.003} C_VEL
LIN {X 0,Y 61.628,Z 660.456,A -85,B 0,C 180,E1 -28719.852,E2 -28719.852} C_VEL
LIN {X 0,Y 57.511,Z 666.076,A -85,B 0,C 180,E1 -28731.51,E2 -28731.51} C_VEL
LIN {X 0,Y 55.381,Z 670.641,A -85,B 0,C 180,E1 -28744.828,E2 -28744.828} C_VEL
LIN {X 0,Y 55.879,Z 674.178,A -85,B 0,C 180,E1 -28758.998,E2 -28758.998} C_VEL
LIN {X 0,Y 58.79,Z 676.53,A -85,B 0,C 180,E1 -28771.431,E2 -28771.431} C_VEL
LIN {X 0,Y 65.533,Z 678.22,A -85,B 0,C 180,E1 -28784.849,E2 -28784.849} C_VEL
LIN {X 0,Y 73.828,Z 678.586,A -85,B 0,C 180,E1 -28794.535,E2 -28794.535} C_VEL
LIN {X 0,Y 84.422,Z 677.82,A -85,B 0,C 180,E1 -28802.537,E2 -28802.537} C_VEL
LIN {X 0,Y 95.692,Z 675.978,A -85,B 0,C 180,E1 -28808.445,E2 -28808.445} C_VEL
LIN {X 0,Y 108.301,Z 672.887,A -85,B 0,C 180,E1 -28813.239,E2 -28813.239} C_VEL
LIN {X 0,Y 121.224,Z 668.617,A -85,B 0,C 180,E1 -28816.888,E2 -28816.888} C_VEL
LIN {X 0,Y 125.569,Z 666.896,A -85,B 0,C 180,E1 -28817.918,E2 -28817.918} C_VEL
LIN {X 0,Y 125.809,Z 666.829,A -85,B 0,C 180,E1 -28818.252,E2 -28818.252} C_VEL
LIN {X 0,Y 113.072,Z 672.107,A -85,B 0,C 180,E1 -28821.196,E2 -28821.196} C_VEL
LIN {X 0,Y 100.828,Z 676.186,A -85,B 0,C 180,E1 -28825.02,E2 -28825.02} C_VEL
LIN {X 0,Y 89.219,Z 679.253,A -85,B 0,C 180,E1 -28829.942,E2 -28829.942} C_VEL
LIN {X 0,Y 78.539,Z 681.356,A -85,B 0,C 180,E1 -28836.351,E2 -28836.351} C_VEL
LIN {X 0,Y 67.875,Z 682.536,A -85,B 0,C 180,E1 -28846.449,E2 -28846.449} C_VEL
LIN {X 0,Y 59.281,Z 682.232,A -85,B 0,C 180,E1 -28861.688,E2 -28861.688} C_VEL
LIN {X 0,Y 56.325,Z 680.85,A -85,B 0,C 180,E1 -28875.546,E2 -28875.546} C_VEL
LIN {X 0,Y 56.288,Z 678.954,A -85,B 0,C 180,E1 -28887.227,E2 -28887.227} C_VEL
LIN {X 0,Y 56.244,Z 677.953,A -85,B 0,C 180,E1 -28891.61,E2 -28891.61} C_VEL
LIN {X 0,Y 56.442,Z 674.191,A -85,B 0,C 180,E1 -28904.417,E2 -28904.417} C_VEL
LIN {X 0,Y 59.445,Z 668.545,A -85,B 0,C 180,E1 -28918.22,E2 -28918.22} C_VEL
LIN {X 0,Y 65.321,Z 661.283,A -85,B 0,C 180,E1 -28930.203,E2 -28930.203} C_VEL
LIN {X 0,Y 72.333,Z 653.44,A -85,B 0,C 180,E1 -28938.847,E2 -28938.847} C_VEL
LIN {X 0,Y 80.551,Z 643.898,A -85,B 0,C 180,E1 -28945.978,E2 -28945.978} C_VEL
LIN {X 0,Y 88.485,Z 634.208,A -85,B 0,C 180,E1 -28950.886,E2 -28950.886} C_VEL
LIN {X 0,Y 96.954,Z 622.682,A -85,B 0,C 180,E1 -28954.968,E2 -28954.968} C_VEL
LIN {X 0,Y 105.126,Z 610.047,A -85,B 0,C 180,E1 -28958.057,E2 -28958.057} C_VEL
LIN {X 0,Y 111.986,Z 597.633,A -85,B 0,C 180,E1 -28960.278,E2 -28960.278} C_VEL
LIN {X 0,Y 118.219,Z 584.315,A -85,B 0,C 180,E1 -28962.018,E2 -28962.018} C_VEL
LIN {X 0,Y 123.673,Z 570.121,A -85,B 0,C 180,E1 -28963.356,E2 -28963.356} C_VEL
LIN {X 0,Y 128.371,Z 554.321,A -85,B 0,C 180,E1 -28964.402,E2 -28964.402} C_VEL
LIN {X 0,Y 131.484,Z 539.384,A -85,B 0,C 180,E1 -28965.142,E2 -28965.142} C_VEL
LIN {X 0,Y 134.856,Z 514.891,A -85,B 0,C 180,E1 -28965.947,E2 -28965.947} C_VEL
LIN {X 0,Y 135.084,Z 511.067,A -85,B 0,C 180,E1 -28966.279,E2 -28966.279} C_VEL
LIN {X 0,Y 134.758,Z 505.652,A -85,B 0,C 180,E1 -28967.265,E2 -28967.265} C_VEL
LIN {X 0,Y 133.895,Z 500.72,A -85,B 0,C 180,E1 -28968.637,E2 -28968.637} C_VEL
LIN {X 0,Y 130.861,Z 488.445,A -85,B 0,C 180,E1 -28973.263,E2 -28973.263} C_VEL
LIN {X 0,Y 128,Z 481.174,A -85,B 0,C 180,E1 -28977.835,E2 -28977.835} C_VEL
LIN {X 0,Y 125.18,Z 474.275,A -85,B 0,C 180,E1 -28983.686,E2 -28983.686} C_VEL
LIN {X 0,Y 123.275,Z 470.035,A -85,B 0,C 180,E1 -28989.077,E2 -28989.077} C_VEL
LIN {X 0,Y 121.991,Z 466.919,A -85,B 0,C 180,E1 -28995.777,E2 -28995.777} C_VEL
LIN {X 0,Y 121.875,Z 466.969,A -85,B 0,C 180,E1 -29004.62,E2 -29004.62} C_VEL
LIN {X 0,Y 122.992,Z 470.355,A -85,B 0,C 180,E1 -29011.39,E2 -29011.39} C_VEL
LIN {X 0,Y 123.616,Z 471.778,A -85,B 0,C 180,E1 -29013.612,E2 -29013.612} C_VEL
LIN {X 0,Y 125.032,Z 474.762,A -85,B 0,C 180,E1 -29017.371,E2 -29017.371} C_VEL
LIN {X 0,Y 127.264,Z 479.638,A -85,B 0,C 180,E1 -29022.052,E2 -29022.052} C_VEL
LIN {X 0,Y 130.326,Z 486.968,A -85,B 0,C 180,E1 -29027.056,E2 -29027.056} C_VEL
LIN {X 0,Y 133.24,Z 494.524,A -85,B 0,C 180,E1 -29031.084,E2 -29031.084} C_VEL
LIN {X 0,Y 133.566,Z 495.41,A -85,B 0,C 180,E1 -29031.495,E2 -29031.495} C_VEL
LIN {X 0,Y 128.186,Z 533.595,A -85,B 0,C 180,E1 -29032.705,E2 -29032.705} C_VEL
LIN {X 0,Y 124.761,Z 549.102,A -85,B 0,C 180,E1 -29033.518,E2 -29033.518} C_VEL
LIN {X 0,Y 120.261,Z 564.042,A -85,B 0,C 180,E1 -29034.658,E2 -29034.658} C_VEL
LIN {X 0,Y 114.466,Z 578.862,A -85,B 0,C 180,E1 -29036.167,E2 -29036.167} C_VEL
LIN {X 0,Y 107.509,Z 593.288,A -85,B 0,C 180,E1 -29038.195,E2 -29038.195} C_VEL
LIN {X 0,Y 100.212,Z 605.934,A -85,B 0,C 180,E1 -29040.601,E2 -29040.601} C_VEL
LIN {X 0,Y 91.88,Z 618.36,A -85,B 0,C 180,E1 -29043.91,E2 -29043.91} C_VEL
LIN {X 0,Y 83.309,Z 629.533,A -85,B 0,C 180,E1 -29048.125,E2 -29048.125} C_VEL
LIN {X 0,Y 74.694,Z 639.592,A -85,B 0,C 180,E1 -29053.607,E2 -29053.607} C_VEL
LIN {X 0,Y 66.332,Z 648.596,A -85,B 0,C 180,E1 -29060.858,E2 -29060.858} C_VEL
LIN {X 0,Y 59.01,Z 656.217,A -85,B 0,C 180,E1 -29070.003,E2 -29070.003} C_VEL
LIN {X 0,Y 53.289,Z 662.538,A -85,B 0,C 180,E1 -29081.413,E2 -29081.413} C_VEL
LIN {X 0,Y 49.438,Z 667.831,A -85,B 0,C 180,E1 -29095.248,E2 -29095.248} C_VEL
LIN {X 0,Y 48.239,Z 672.646,A -85,B 0,C 180,E1 -29113.239,E2 -29113.239} C_VEL
LIN {X 0,Y 50.155,Z 675.483,A -85,B 0,C 180,E1 -29127.227,E2 -29127.227} C_VEL
LIN {X 0,Y 53.369,Z 677.084,A -85,B 0,C 180,E1 -29137.201,E2 -29137.201} C_VEL
LIN {X 0,Y 57.958,Z 678.209,A -85,B 0,C 180,E1 -29145.962,E2 -29145.962} C_VEL
LIN {X 0,Y 63.821,Z 678.884,A -85,B 0,C 180,E1 -29153.675,E2 -29153.675} C_VEL
LIN {X 0,Y 70.543,Z 679.058,A -85,B 0,C 180,E1 -29159.998,E2 -29159.998} C_VEL
LIN {X 0,Y 77.974,Z 678.729,A -85,B 0,C 180,E1 -29165.169,E2 -29165.169} C_VEL
LIN {X 0,Y 85.843,Z 677.87,A -85,B 0,C 180,E1 -29169.422,E2 -29169.422} C_VEL
LIN {X 0,Y 94.152,Z 676.498,A -85,B 0,C 180,E1 -29172.939,E2 -29172.939} C_VEL
LIN {X 0,Y 108.724,Z 673.034,A -85,B 0,C 180,E1 -29177.589,E2 -29177.589} C_VEL
LIN {X 0,Y 105.985,Z 674.022,A -85,B 0,C 180,E1 -29178.917,E2 -29178.917} C_VEL
LIN {X 0,Y 91.87,Z 677.92,A -85,B 0,C 180,E1 -29183.361,E2 -29183.361} C_VEL
LIN {X 0,Y 80.05,Z 680.265,A -85,B 0,C 180,E1 -29188.6,E2 -29188.6} C_VEL
LIN {X 0,Y 69.294,Z 681.696,A -85,B 0,C 180,E1 -29195.764,E2 -29195.764} C_VEL
LIN {X 0,Y 60.085,Z 682.126,A -85,B 0,C 180,E1 -29205.424,E2 -29205.424} C_VEL
LIN {X 0,Y 53.095,Z 681.574,A -85,B 0,C 180,E1 -29218.026,E2 -29218.026} C_VEL
LIN {X 0,Y 49.447,Z 680.076,A -85,B 0,C 180,E1 -29233.481,E2 -29233.481} C_VEL
LIN {X 0,Y 49.249,Z 677.956,A -85,B 0,C 180,E1 -29247.29,E2 -29247.29} C_VEL
LIN {X 0,Y 49.203,Z 677.197,A -85,B 0,C 180,E1 -29251.124,E2 -29251.124} C_VEL
LIN {X 0,Y 49.553,Z 673.081,A -85,B 0,C 180,E1 -29266.475,E2 -29266.475} C_VEL
LIN {X 0,Y 53.24,Z 667.223,A -85,B 0,C 180,E1 -29281.868,E2 -29281.868} C_VEL
LIN {X 0,Y 60.03,Z 659.736,A -85,B 0,C 180,E1 -29294.62,E2 -29294.62} C_VEL
LIN {X 0,Y 67.817,Z 651.636,A -85,B 0,C 180,E1 -29303.427,E2 -29303.427} C_VEL
LIN {X 0,Y 76.763,Z 641.812,A -85,B 0,C 180,E1 -29310.427,E2 -29310.427} C_VEL
LIN {X 0,Y 85.227,Z 631.798,A -85,B 0,C 180,E1 -29315.101,E2 -29315.101} C_VEL
LIN {X 0,Y 94.145,Z 619.884,A -85,B 0,C 180,E1 -29318.923,E2 -29318.923} C_VEL
LIN {X 0,Y 101.878,Z 608.083,A -85,B 0,C 180,E1 -29321.532,E2 -29321.532} C_VEL
LIN {X 0,Y 108.977,Z 595.367,A -85,B 0,C 180,E1 -29323.59,E2 -29323.59} C_VEL
LIN {X 0,Y 115.392,Z 581.628,A -85,B 0,C 180,E1 -29325.204,E2 -29325.204} C_VEL
LIN {X 0,Y 121.234,Z 566.176,A -85,B 0,C 180,E1 -29326.455,E2 -29326.455} C_VEL
LIN {X 0,Y 125.599,Z 550.857,A -85,B 0,C 180,E1 -29327.344,E2 -29327.344} C_VEL
LIN {X 0,Y 128.652,Z 535.252,A -85,B 0,C 180,E1 -29328.002,E2 -29328.002} C_VEL
LIN {X 0,Y 133.527,Z 499.112,A -85,B 0,C 180,E1 -29329.164,E2 -29329.164} C_VEL
LIN {X 0,Y 131.214,Z 489.884,A -85,B 0,C 180,E1 -29332.667,E2 -29332.667} C_VEL
LIN {X 0,Y 130.861,Z 488.445,A -85,B 0,C 180,E1 -29333.263,E2 -29333.263} C_VEL
LIN {X 0,Y 130.1,Z 485.935,A -85,B 0,C 180,E1 -29334.513,E2 -29334.513} C_VEL
LIN {X 0,Y 129.099,Z 484.138,A -85,B 0,C 180,E1 -29335.974,E2 -29335.974} C_VEL
LIN {X 0,Y 127.946,Z 482.9,A -85,B 0,C 180,E1 -29337.573,E2 -29337.573} C_VEL
LIN {X 0,Y 123.66,Z 480.293,A -85,B 0,C 180,E1 -29344.723,E2 -29344.723} C_VEL
LIN {X 0,Y 122.895,Z 479.266,A -85,B 0,C 180,E1 -29346.559,E2 -29346.559} C_VEL
LIN {X 0,Y 121.921,Z 476.803,A -85,B 0,C 180,E1 -29349.96,E2 -29349.96} C_VEL
LIN {X 0,Y 120.9,Z 473.928,A -85,B 0,C 180,E1 -29355.924,E2 -29355.924} C_VEL
LIN {X 0,Y 120.752,Z 473.913,A -85,B 0,C 180,E1 -29364.044,E2 -29364.044} C_VEL
LIN {X 0,Y 122.12,Z 478.144,A -85,B 0,C 180,E1 -29372.33,E2 -29372.33} C_VEL
LIN {X 0,Y 123.592,Z 481.689,A -85,B 0,C 180,E1 -29376.752,E2 -29376.752} C_VEL
LIN {X 0,Y 125.614,Z 486.536,A -85,B 0,C 180,E1 -29381.287,E2 -29381.287} C_VEL
LIN {X 0,Y 128.113,Z 493.093,A -85,B 0,C 180,E1 -29385.746,E2 -29385.746} C_VEL
LIN {X 0,Y 130.061,Z 498.423,A -85,B 0,C 180,E1 -29388.734,E2 -29388.734} C_VEL
LIN {X 0,Y 128.041,Z 513.505,A -85,B 0,C 180,E1 -29389.217,E2 -29389.217} C_VEL
LIN {X 0,Y 124.687,Z 535.362,A -85,B 0,C 180,E1 -29389.889,E2 -29389.889} C_VEL
LIN {X 0,Y 121.063,Z 550.944,A -85,B 0,C 180,E1 -29390.696,E2 -29390.696} C_VEL
LIN {X 0,Y 116.363,Z 565.67,A -85,B 0,C 180,E1 -29391.738,E2 -29391.738} C_VEL
LIN {X 0,Y 110.102,Z 580.96,A -85,B 0,C 180,E1 -29393.245,E2 -29393.245} C_VEL
LIN {X 0,Y 103.187,Z 594.652,A -85,B 0,C 180,E1 -29395.095,E2 -29395.095} C_VEL
LIN {X 0,Y 95.036,Z 608.091,A -85,B 0,C 180,E1 -29397.581,E2 -29397.581} C_VEL
LIN {X 0,Y 86.422,Z 620.224,A -85,B 0,C 180,E1 -29400.798,E2 -29400.798} C_VEL
LIN {X 0,Y 76.948,Z 631.775,A -85,B 0,C 180,E1 -29405.247,E2 -29405.247} C_VEL
LIN {X 0,Y 68.473,Z 640.992,A -85,B 0,C 180,E1 -29410.517,E2 -29410.517} C_VEL
LIN {X 0,Y 58.926,Z 650.445,A -85,B 0,C 180,E1 -29418.751,E2 -29418.751} C_VEL
LIN {X 0,Y 50.635,Z 658.408,A -85,B 0,C 180,E1 -29430.004,E2 -29430.004} C_VEL
LIN {X 0,Y 45.205,Z 664.118,A -85,B 0,C 180,E1 -29442.519,E2 -29442.519} C_VEL
LIN {X 0,Y 41.496,Z 669.592,A -85,B 0,C 180,E1 -29460.542,E2 -29460.542} C_VEL
LIN {X 0,Y 41.379,Z 673.175,A -85,B 0,C 180,E1 -29477.199,E2 -29477.199} C_VEL
LIN {X 0,Y 45.664,Z 676.627,A -85,B 0,C 180,E1 -29497.446,E2 -29497.446} C_VEL
LIN {X 0,Y 53.773,Z 678.667,A -85,B 0,C 180,E1 -29512.487,E2 -29512.487} C_VEL
LIN {X 0,Y 63.315,Z 679.509,A -85,B 0,C 180,E1 -29522.486,E2 -29522.486} C_VEL
LIN {X 0,Y 76.009,Z 679.224,A -85,B 0,C 180,E1 -29530.655,E2 -29530.655} C_VEL
LIN {X 0,Y 87.586,Z 677.933,A -85,B 0,C 180,E1 -29535.65,E2 -29535.65} C_VEL
LIN {X 0,Y 93.219,Z 677.017,A -85,B 0,C 180,E1 -29537.55,E2 -29537.55} C_VEL
LIN {X 0,Y 89.28,Z 677.944,A -85,B 0,C 180,E1 -29539.151,E2 -29539.151} C_VEL
LIN {X 0,Y 76.883,Z 680.125,A -85,B 0,C 180,E1 -29543.914,E2 -29543.914} C_VEL
LIN {X 0,Y 65.368,Z 681.332,A -85,B 0,C 180,E1 -29550.665,E2 -29550.665} C_VEL
LIN {X 0,Y 55.204,Z 681.64,A -85,B 0,C 180,E1 -29560.19,E2 -29560.19} C_VEL
LIN {X 0,Y 47.184,Z 680.911,A -85,B 0,C 180,E1 -29573.426,E2 -29573.426} C_VEL
LIN {X 0,Y 42.665,Z 679.226,A -85,B 0,C 180,E1 -29590.76,E2 -29590.76} C_VEL
LIN {X 0,Y 42.218,Z 676.97,A -85,B 0,C 180,E1 -29607.134,E2 -29607.134} C_VEL
LIN {X 0,Y 42.167,Z 676.366,A -85,B 0,C 180,E1 -29610.478,E2 -29610.478} C_VEL
LIN {X 0,Y 42.765,Z 671.939,A -85,B 0,C 180,E1 -29629.184,E2 -29629.184} C_VEL
LIN {X 0,Y 47.302,Z 665.875,A -85,B 0,C 180,E1 -29646.458,E2 -29646.458} C_VEL
LIN {X 0,Y 55.154,Z 658.17,A -85,B 0,C 180,E1 -29659.862,E2 -29659.862} C_VEL
LIN {X 0,Y 63.785,Z 649.829,A -85,B 0,C 180,E1 -29668.635,E2 -29668.635} C_VEL
LIN {X 0,Y 73.46,Z 639.704,A -85,B 0,C 180,E1 -29675.345,E2 -29675.345} C_VEL
LIN {X 0,Y 82.463,Z 629.388,A -85,B 0,C 180,E1 -29679.627,E2 -29679.627} C_VEL
LIN {X 0,Y 91.818,Z 617.093,A -85,B 0,C 180,E1 -29683.087,E2 -29683.087} C_VEL
LIN {X 0,Y 100.651,Z 603.444,A -85,B 0,C 180,E1 -29685.649,E2 -29685.649} C_VEL
LIN {X 0,Y 107.981,Z 589.776,A -85,B 0,C 180,E1 -29687.489,E2 -29687.489} C_VEL
LIN {X 0,Y 114.189,Z 575.856,A -85,B 0,C 180,E1 -29688.778,E2 -29688.778} C_VEL
LIN {X 0,Y 119.332,Z 561.348,A -85,B 0,C 180,E1 -29689.747,E2 -29689.747} C_VEL
LIN {X 0,Y 123.374,Z 546.251,A -85,B 0,C 180,E1 -29690.437,E2 -29690.437} C_VEL
LIN {X 0,Y 126.24,Z 529.896,A -85,B 0,C 180,E1 -29691.007,E2 -29691.007} C_VEL
LIN {X 0,Y 130.096,Z 501.68,A -85,B 0,C 180,E1 -29691.838,E2 -29691.838} C_VEL
LIN {X 0,Y 128.177,Z 493.131,A -85,B 0,C 180,E1 -29695.346,E2 -29695.346} C_VEL
LIN {X 0,Y 125.273,Z 485.391,A -85,B 0,C 180,E1 -29700.623,E2 -29700.623} C_VEL
LIN {X 0,Y 123.195,Z 479.863,A -85,B 0,C 180,E1 -29705.743,E2 -29705.743} C_VEL
LIN {X 0,Y 122.895,Z 479.266,A -85,B 0,C 180,E1 -29706.559,E2 -29706.559} C_VEL
LIN {X 0,Y 121.953,Z 478.213,A -85,B 0,C 180,E1 -29709.248,E2 -29709.248} C_VEL
LIN {X 0,Y 121.083,Z 478.317,A -85,B 0,C 180,E1 -29712.029,E2 -29712.029} C_VEL
LIN {X 0,Y 119.585,Z 480.61,A -85,B 0,C 180,E1 -29719.642,E2 -29719.642} C_VEL
LIN {X 0,Y 119.54,Z 480.859,A -85,B 0,C 180,E1 -29721.586,E2 -29721.586} C_VEL
LIN {X 0,Y 119.64,Z 481.18,A -85,B 0,C 180,E1 -29724.041,E2 -29724.041} C_VEL
LIN {X 0,Y 120.751,Z 484.83,A -85,B 0,C 180,E1 -29731.369,E2 -29731.369} C_VEL
LIN {X 0,Y 122.039,Z 488.346,A -85,B 0,C 180,E1 -29735.785,E2 -29735.785} C_VEL
LIN {X 0,Y 123.915,Z 493.223,A -85,B 0,C 180,E1 -29740.345,E2 -29740.345} C_VEL
LIN {X 0,Y 126.318,Z 500.296,A -85,B 0,C 180,E1 -29745.047,E2 -29745.047} C_VEL
LIN {X 0,Y 126.848,Z 501.798,A -85,B 0,C 180,E1 -29745.926,E2 -29745.926} C_VEL
LIN {X 0,Y 122.226,Z 533.453,A -85,B 0,C 180,E1 -29746.82,E2 -29746.82} C_VEL
LIN {X 0,Y 118.631,Z 549.19,A -85,B 0,C 180,E1 -29747.495,E2 -29747.495} C_VEL
LIN {X 0,Y 113.881,Z 564.302,A -85,B 0,C 180,E1 -29748.452,E2 -29748.452} C_VEL
LIN {X 0,Y 108.367,Z 577.935,A -85,B 0,C 180,E1 -29749.571,E2 -29749.571} C_VEL
LIN {X 0,Y 101.084,Z 592.533,A -85,B 0,C 180,E1 -29751.266,E2 -29751.266} C_VEL
LIN {X 0,Y 92.827,Z 606.1,A -85,B 0,C 180,E1 -29753.403,E2 -29753.403} C_VEL
LIN {X 0,Y 84.023,Z 618.39,A -85,B 0,C 180,E1 -29756.211,E2 -29756.211} C_VEL
LIN {X 0,Y 74.19,Z 630.169,A -85,B 0,C 180,E1 -29760.179,E2 -29760.179} C_VEL
LIN {X 0,Y 64.08,Z 640.75,A -85,B 0,C 180,E1 -29765.707,E2 -29765.707} C_VEL
LIN {X 0,Y 54.457,Z 649.724,A -85,B 0,C 180,E1 -29773.123,E2 -29773.123} C_VEL
LIN {X 0,Y 45.925,Z 657.285,A -85,B 0,C 180,E1 -29783.413,E2 -29783.413} C_VEL
LIN {X 0,Y 40.008,Z 662.622,A -85,B 0,C 180,E1 -29795.038,E2 -29795.038} C_VEL
LIN {X 0,Y 35.176,Z 668.095,A -85,B 0,C 180,E1 -29813.558,E2 -29813.558} C_VEL
LIN {X 0,Y 34.133,Z 672.501,A -85,B 0,C 180,E1 -29835.54,E2 -29835.54} C_VEL
LIN {X 0,Y 38.134,Z 676.12,A -85,B 0,C 180,E1 -29858.367,E2 -29858.367} C_VEL
LIN {X 0,Y 43.612,Z 677.919,A -85,B 0,C 180,E1 -29870.723,E2 -29870.723} C_VEL
LIN {X 0,Y 50.369,Z 679.121,A -85,B 0,C 180,E1 -29879.997,E2 -29879.997} C_VEL
LIN {X 0,Y 57.934,Z 679.809,A -85,B 0,C 180,E1 -29886.965,E2 -29886.965} C_VEL
LIN {X 0,Y 66.145,Z 680.007,A -85,B 0,C 180,E1 -29892.267,E2 -29892.267} C_VEL
LIN {X 0,Y 76.644,Z 679.571,A -85,B 0,C 180,E1 -29897.112,E2 -29897.112} C_VEL
LIN {X 0,Y 74.275,Z 679.944,A -85,B 0,C 180,E1 -29898.87,E2 -29898.87} C_VEL
LIN {X 0,Y 62.016,Z 680.971,A -85,B 0,C 180,E1 -29904.953,E2 -29904.953} C_VEL
LIN {X 0,Y 50.871,Z 681.068,A -85,B 0,C 180,E1 -29914.006,E2 -29914.006} C_VEL
LIN {X 0,Y 41.665,Z 680.236,A -85,B 0,C 180,E1 -29927.562,E2 -29927.562} C_VEL
LIN {X 0,Y 36.025,Z 678.364,A -85,B 0,C 180,E1 -29947.029,E2 -29947.029} C_VEL
LIN {X 0,Y 35.182,Z 675.917,A -85,B 0,C 180,E1 -29967.121,E2 -29967.121} C_VEL
LIN {X 0,Y 35.392,Z 672.016,A -85,B 0,C 180,E1 -29987.324,E2 -29987.324} C_VEL
LIN {X 0,Y 39.964,Z 666.118,A -85,B 0,C 180,E1 -30007.983,E2 -30007.983} C_VEL
LIN {X 0,Y 48.339,Z 658.593,A -85,B 0,C 180,E1 -30023.091,E2 -30023.091} C_VEL
LIN {X 0,Y 57.54,Z 650.454,A -85,B 0,C 180,E1 -30032.31,E2 -30032.31} C_VEL
LIN {X 0,Y 67.715,Z 640.569,A -85,B 0,C 180,E1 -30039.075,E2 -30039.075} C_VEL
LIN {X 0,Y 77.065,Z 630.513,A -85,B 0,C 180,E1 -30043.239,E2 -30043.239} C_VEL
LIN {X 0,Y 86.718,Z 618.536,A -85,B 0,C 180,E1 -30046.53,E2 -30046.53} C_VEL
LIN {X 0,Y 94.951,Z 606.634,A -85,B 0,C 180,E1 -30048.723,E2 -30048.723} C_VEL
LIN {X 0,Y 102.459,Z 593.817,A -85,B 0,C 180,E1 -30050.399,E2 -30050.399} C_VEL
LIN {X 0,Y 109.199,Z 579.946,A -85,B 0,C 180,E1 -30051.688,E2 -30051.688} C_VEL
LIN {X 0,Y 115.097,Z 564.821,A -85,B 0,C 180,E1 -30052.643,E2 -30052.643} C_VEL
LIN {X 0,Y 119.666,Z 549.25,A -85,B 0,C 180,E1 -30053.337,E2 -30053.337} C_VEL
LIN {X 0,Y 122.853,Z 533.137,A -85,B 0,C 180,E1 -30053.897,E2 -30053.897} C_VEL
LIN {X 0,Y 126.949,Z 504.325,A -85,B 0,C 180,E1 -30054.659,E2 -30054.659} C_VEL
LIN {X 0,Y 125.569,Z 498.011,A -85,B 0,C 180,E1 -30057.465,E2 -30057.465} C_VEL
LIN {X 0,Y 123.272,Z 491.176,A -85,B 0,C 180,E1 -30062.348,E2 -30062.348} C_VEL
LIN {X 0,Y 121.643,Z 486.378,A -85,B 0,C 180,E1 -30066.865,E2 -30066.865} C_VEL
LIN {X 0,Y 120.58,Z 483.489,A -85,B 0,C 180,E1 -30070.949,E2 -30070.949} C_VEL
LIN {X 0,Y 119.785,Z 481.054,A -85,B 0,C 180,E1 -30076.076,E2 -30076.076} C_VEL
LIN {X 0,Y 119.54,Z 480.859,A -85,B 0,C 180,E1 -30081.586,E2 -30081.586} C_VEL
LIN {X 0,Y 119.566,Z 481.366,A -85,B 0,C 180,E1 -30083.445,E2 -30083.445} C_VEL
LIN {X 0,Y 119.602,Z 483.418,A -85,B 0,C 180,E1 -30086.099,E2 -30086.099} C_VEL
LIN {X 0,Y 119.669,Z 486.419,A -85,B 0,C 180,E1 -30088.57,E2 -30088.57} C_VEL
LIN {X 0,Y 120.201,Z 493.338,A -85,B 0,C 180,E1 -30093.446,E2 -30093.446} C_VEL
LIN {X 0,Y 120.639,Z 495.303,A -85,B 0,C 180,E1 -30095.147,E2 -30095.147} C_VEL
LIN {X 0,Y 122.187,Z 499.832,A -85,B 0,C 180,E1 -30099.251,E2 -30099.251} C_VEL
LIN {X 0,Y 123.867,Z 505.36,A -85,B 0,C 180,E1 -30103.037,E2 -30103.037} C_VEL
LIN {X 0,Y 119.37,Z 534.676,A -85,B 0,C 180,E1 -30103.714,E2 -30103.714} C_VEL
LIN {X 0,Y 115.755,Z 550.066,A -85,B 0,C 180,E1 -30104.335,E2 -30104.335} C_VEL
LIN {X 0,Y 110.856,Z 565.116,A -85,B 0,C 180,E1 -30105.149,E2 -30105.149} C_VEL
LIN {X 0,Y 104.84,Z 579.517,A -85,B 0,C 180,E1 -30106.237,E2 -30106.237} C_VEL
LIN {X 0,Y 97.773,Z 593.208,A -85,B 0,C 180,E1 -30107.635,E2 -30107.635} C_VEL
LIN {X 0,Y 89.166,Z 606.907,A -85,B 0,C 180,E1 -30109.534,E2 -30109.534} C_VEL
LIN {X 0,Y 80.038,Z 619.2,A -85,B 0,C 180,E1 -30112.076,E2 -30112.076} C_VEL
LIN {X 0,Y 70.938,Z 629.735,A -85,B 0,C 180,E1 -30115.215,E2 -30115.215} C_VEL
LIN {X 0,Y 60.169,Z 640.533,A -85,B 0,C 180,E1 -30120.24,E2 -30120.24} C_VEL
LIN {X 0,Y 49.843,Z 649.588,A -85,B 0,C 180,E1 -30127.189,E2 -30127.189} C_VEL
LIN {X 0,Y 40.307,Z 657.291,A -85,B 0,C 180,E1 -30137.587,E2 -30137.587} C_VEL
LIN {X 0,Y 32.474,Z 663.616,A -85,B 0,C 180,E1 -30153.107,E2 -30153.107} C_VEL
LIN {X 0,Y 28.016,Z 668.255,A -85,B 0,C 180,E1 -30172.48,E2 -30172.48} C_VEL
LIN {X 0,Y 27.331,Z 672.765,A -85,B 0,C 180,E1 -30200.494,E2 -30200.494} C_VEL
LIN {X 0,Y 33.339,Z 676.562,A -85,B 0,C 180,E1 -30227.826,E2 -30227.826} C_VEL
LIN {X 0,Y 42.215,Z 678.725,A -85,B 0,C 180,E1 -30242.612,E2 -30242.612} C_VEL
LIN {X 0,Y 56.318,Z 680.27,A -85,B 0,C 180,E1 -30254.45,E2 -30254.45} C_VEL
LIN {X 0,Y 60.438,Z 680.46,A -85,B 0,C 180,E1 -30256.681,E2 -30256.681} C_VEL
LIN {X 0,Y 59.352,Z 680.596,A -85,B 0,C 180,E1 -30258.675,E2 -30258.675} C_VEL
LIN {X 0,Y 47.232,Z 680.486,A -85,B 0,C 180,E1 -30266.768,E2 -30266.768} C_VEL
LIN {X 0,Y 36.718,Z 679.471,A -85,B 0,C 180,E1 -30280.03,E2 -30280.03} C_VEL
LIN {X 0,Y 29.611,Z 677.489,A -85,B 0,C 180,E1 -30301.654,E2 -30301.654} C_VEL
LIN {X 0,Y 28.122,Z 674.599,A -85,B 0,C 180,E1 -30328.268,E2 -30328.268} C_VEL
LIN {X 0,Y 28.651,Z 670.825,A -85,B 0,C 180,E1 -30351.582,E2 -30351.582} C_VEL
LIN {X 0,Y 34.604,Z 664.719,A -85,B 0,C 180,E1 -30375.297,E2 -30375.297} C_VEL
LIN {X 0,Y 43.061,Z 657.991,A -85,B 0,C 180,E1 -30388.958,E2 -30388.958} C_VEL
LIN {X 0,Y 54.565,Z 648.53,A -85,B 0,C 180,E1 -30399.027,E2 -30399.027} C_VEL
LIN {X 0,Y 65.487,Z 638.309,A -85,B 0,C 180,E1 -30404.977,E2 -30404.977} C_VEL
LIN {X 0,Y 75.313,Z 627.956,A -85,B 0,C 180,E1 -30408.461,E2 -30408.461} C_VEL
LIN {X 0,Y 85.337,Z 615.526,A -85,B 0,C 180,E1 -30411.201,E2 -30411.201} C_VEL
LIN {X 0,Y 93.818,Z 603.146,A -85,B 0,C 180,E1 -30412.994,E2 -30412.994} C_VEL
LIN {X 0,Y 101.51,Z 589.643,A -85,B 0,C 180,E1 -30414.394,E2 -30414.394} C_VEL
LIN {X 0,Y 108.397,Z 574.829,A -85,B 0,C 180,E1 -30415.426,E2 -30415.426} C_VEL
LIN {X 0,Y 113.567,Z 560.825,A -85,B 0,C 180,E1 -30416.12,E2 -30416.12} C_VEL
LIN {X 0,Y 117.85,Z 545.373,A -85,B 0,C 180,E1 -30416.643,E2 -30416.643} C_VEL
LIN {X 0,Y 120.907,Z 528.547,A -85,B 0,C 180,E1 -30417.093,E2 -30417.093} C_VEL
LIN {X 0,Y 123.976,Z 506.876,A -85,B 0,C 180,E1 -30417.66,E2 -30417.66} C_VEL
LIN {X 0,Y 123.215,Z 503.231,A -85,B 0,C 180,E1 -30419.465,E2 -30419.465} C_VEL
LIN {X 0,Y 121.467,Z 497.241,A -85,B 0,C 180,E1 -30423.859,E2 -30423.859} C_VEL
LIN {X 0,Y 120.098,Z 492.772,A -85,B 0,C 180,E1 -30428.165,E2 -30428.165} C_VEL
LIN {X 0,Y 119.273,Z 490.193,A -85,B 0,C 180,E1 -30431.961,E2 -30431.961} C_VEL
LIN {X 0,Y 118.595,Z 487.889,A -85,B 0,C 180,E1 -30437.237,E2 -30437.237} C_VEL
LIN {X 0,Y 118.532,Z 488.037,A -85,B 0,C 180,E1 -30443.359,E2 -30443.359} C_VEL
LIN {X 0,Y 119.48,Z 491.746,A -85,B 0,C 180,E1 -30450.728,E2 -30450.728} C_VEL
LIN {X 0,Y 120.598,Z 495.169,A -85,B 0,C 180,E1 -30455.015,E2 -30455.015} C_VEL
LIN {X 0,Y 120.639,Z 495.303,A -85,B 0,C 180,E1 -30455.147,E2 -30455.147} C_VEL
LIN {X 0,Y 121.075,Z 497.634,A -85,B 0,C 180,E1 -30456.731,E2 -30456.731} C_VEL
LIN {X 0,Y 121.295,Z 500.768,A -85,B 0,C 180,E1 -30458.001,E2 -30458.001} C_VEL
LIN {X 0,Y 121.244,Z 505.715,A -85,B 0,C 180,E1 -30459.225,E2 -30459.225} C_VEL
LIN {X 0,Y 120.803,Z 511.149,A -85,B 0,C 180,E1 -30459.922,E2 -30459.922} C_VEL
LIN {X 0,Y 120.437,Z 513.938,A -85,B 0,C 180,E1 -30460.05,E2 -30460.05} C_VEL
LIN {X 0,Y 116.891,Z 535.92,A -85,B 0,C 180,E1 -30460.49,E2 -30460.49} C_VEL
LIN {X 0,Y 113.172,Z 551.178,A -85,B 0,C 180,E1 -30461.025,E2 -30461.025} C_VEL
LIN {X 0,Y 108.216,Z 565.954,A -85,B 0,C 180,E1 -30461.684,E2 -30461.684} C_VEL
LIN {X 0,Y 102.518,Z 579.38,A -85,B 0,C 180,E1 -30462.53,E2 -30462.53} C_VEL
LIN {X 0,Y 94.861,Z 593.868,A -85,B 0,C 180,E1 -30463.754,E2 -30463.754} C_VEL
LIN {X 0,Y 86.206,Z 607.304,A -85,B 0,C 180,E1 -30465.322,E2 -30465.322} C_VEL
LIN {X 0,Y 76.673,Z 619.73,A -85,B 0,C 180,E1 -30467.481,E2 -30467.481} C_VEL
LIN {X 0,Y 66.234,Z 631.234,A -85,B 0,C 180,E1 -30470.461,E2 -30470.461} C_VEL
LIN {X 0,Y 55.05,Z 641.78,A -85,B 0,C 180,E1 -30474.94,E2 -30474.94} C_VEL
LIN {X 0,Y 44.119,Z 650.696,A -85,B 0,C 180,E1 -30481.457,E2 -30481.457} C_VEL
LIN {X 0,Y 33.821,Z 658.246,A -85,B 0,C 180,E1 -30491.844,E2 -30491.844} C_VEL
LIN {X 0,Y 24.99,Z 664.603,A -85,B 0,C 180,E1 -30510.007,E2 -30510.007} C_VEL
LIN {X 0,Y 20.975,Z 668.267,A -85,B 0,C 180,E1 -30529.585,E2 -30529.585} C_VEL
LIN {X 0,Y 20.749,Z 672.897,A -85,B 0,C 180,E1 -30567.88,E2 -30567.88} C_VEL
LIN {X 0,Y 29.731,Z 676.98,A -85,B 0,C 180,E1 -30599.995,E2 -30599.995} C_VEL
LIN {X 0,Y 43.798,Z 679.7,A -85,B 0,C 180,E1 -30615.664,E2 -30615.664} C_VEL
LIN {X 0,Y 44.825,Z 679.922,A -85,B 0,C 180,E1 -30618.271,E2 -30618.271} C_VEL
LIN {X 0,Y 32.594,Z 678.673,A -85,B 0,C 180,E1 -30630.391,E2 -30630.391} C_VEL
LIN {X 0,Y 23.603,Z 676.533,A -85,B 0,C 180,E1 -30653.441,E2 -30653.441} C_VEL
LIN {X 0,Y 21.363,Z 675.079,A -85,B 0,C 180,E1 -30670.784,E2 -30670.784} C_VEL
LIN {X 0,Y 20.913,Z 673.261,A -85,B 0,C 180,E1 -30689.991,E2 -30689.991} C_VEL
LIN {X 0,Y 23.621,Z 668.084,A -85,B 0,C 180,E1 -30726.508,E2 -30726.508} C_VEL
LIN {X 0,Y 32.635,Z 661.328,A -85,B 0,C 180,E1 -30749.463,E2 -30749.463} C_VEL
LIN {X 0,Y 43.026,Z 653.87,A -85,B 0,C 180,E1 -30760.534,E2 -30760.534} C_VEL
LIN {X 0,Y 54.049,Z 645.057,A -85,B 0,C 180,E1 -30767.203,E2 -30767.203} C_VEL
LIN {X 0,Y 64.01,Z 635.926,A -85,B 0,C 180,E1 -30771.154,E2 -30771.154} C_VEL
LIN {X 0,Y 74.212,Z 625.213,A -85,B 0,C 180,E1 -30773.893,E2 -30773.893} C_VEL
LIN {X 0,Y 84.538,Z 612.318,A -85,B 0,C 180,E1 -30776.006,E2 -30776.006} C_VEL
LIN {X 0,Y 93.216,Z 599.362,A -85,B 0,C 180,E1 -30777.37,E2 -30777.37} C_VEL
LIN {X 0,Y 101.063,Z 585.129,A -85,B 0,C 180,E1 -30778.417,E2 -30778.417} C_VEL
LIN {X 0,Y 107.626,Z 570.392,A -85,B 0,C 180,E1 -30779.119,E2 -30779.119} C_VEL
LIN {X 0,Y 112.791,Z 555.351,A -85,B 0,C 180,E1 -30779.656,E2 -30779.656} C_VEL
LIN {X 0,Y 116.411,Z 540.96,A -85,B 0,C 180,E1 -30780.035,E2 -30780.035} C_VEL
LIN {X 0,Y 120.136,Z 518.102,A -85,B 0,C 180,E1 -30780.502,E2 -30780.502} C_VEL
LIN {X 0,Y 121.314,Z 509.659,A -85,B 0,C 180,E1 -30780.761,E2 -30780.761} C_VEL
LIN {X 0,Y 119.89,Z 504.035,A -85,B 0,C 180,E1 -30784.785,E2 -30784.785} C_VEL
LIN {X 0,Y 118.668,Z 499.331,A -85,B 0,C 180,E1 -30789.274,E2 -30789.274} C_VEL
LIN {X 0,Y 118.068,Z 497.1,A -85,B 0,C 180,E1 -30792.507,E2 -30792.507} C_VEL
LIN {X 0,Y 117.509,Z 494.878,A -85,B 0,C 180,E1 -30797.401,E2 -30797.401} C_VEL
LIN {X 0,Y 117.429,Z 495.018,A -85,B 0,C 180,E1 -30802.817,E2 -30802.817} C_VEL
LIN {X 0,Y 118.162,Z 498.447,A -85,B 0,C 180,E1 -30809.779,E2 -30809.779} C_VEL
LIN {X 0,Y 118.985,Z 501.371,A -85,B 0,C 180,E1 -30813.535,E2 -30813.535} C_VEL
LIN {X 0,Y 120.325,Z 505.831,A -85,B 0,C 180,E1 -30817.715,E2 -30817.715} C_VEL
LIN {X 0,Y 121.138,Z 508.842,A -85,B 0,C 180,E1 -30819.876,E2 -30819.876} C_VEL
LIN {X 0,Y 120.437,Z 513.938,A -85,B 0,C 180,E1 -30820.05,E2 -30820.05} C_VEL
LIN {X 0,Y 119.4,Z 519.739,A -85,B 0,C 180,E1 -30819.853,E2 -30819.853} C_VEL
LIN {X 0,Y 114.633,Z 538.398,A -85,B 0,C 180,E1 -30817.535,E2 -30817.535} C_VEL
LIN {X 0,Y 113.094,Z 544.093,A -85,B 0,C 180,E1 -30817.31,E2 -30817.31} C_VEL
LIN {X 0,Y 108.596,Z 559.402,A -85,B 0,C 180,E1 -30817.844,E2 -30817.844} C_VEL
LIN {X 0,Y 102.747,Z 574.283,A -85,B 0,C 180,E1 -30818.428,E2 -30818.428} C_VEL
LIN {X 0,Y 95.35,Z 589.193,A -85,B 0,C 180,E1 -30819.295,E2 -30819.295} C_VEL
LIN {X 0,Y 86.839,Z 603.073,A -85,B 0,C 180,E1 -30820.352,E2 -30820.352} C_VEL
LIN {X 0,Y 77.75,Z 615.444,A -85,B 0,C 180,E1 -30821.781,E2 -30821.781} C_VEL
LIN {X 0,Y 67.955,Z 626.699,A -85,B 0,C 180,E1 -30823.622,E2 -30823.622} C_VEL
LIN {X 0,Y 57.731,Z 636.765,A -85,B 0,C 180,E1 -30826.201,E2 -30826.201} C_VEL
LIN {X 0,Y 47.01,Z 645.844,A -85,B 0,C 180,E1 -30829.973,E2 -30829.973} C_VEL
LIN {X 0,Y 35.049,Z 654.53,A -85,B 0,C 180,E1 -30836.698,E2 -30836.698} C_VEL
LIN {X 0,Y 24.135,Z 661.464,A -85,B 0,C 180,E1 -30848.663,E2 -30848.663} C_VEL
LIN {X 0,Y 16.21,Z 666.442,A -85,B 0,C 180,E1 -30870.011,E2 -30870.011} C_VEL
LIN {X 0,Y 12.736,Z 669.948,A -85,B 0,C 180,E1 -30903.508,E2 -30903.508} C_VEL
LIN {X 0,Y 14.823,Z 673.001,A -85,B 0,C 180,E1 -30941.523,E2 -30941.523} C_VEL
LIN {X 0,Y 21.152,Z 675.622,A -85,B 0,C 180,E1 -30964.491,E2 -30964.491} C_VEL
LIN {X 0,Y 29.28,Z 677.746,A -85,B 0,C 180,E1 -30976.217,E2 -30976.217} C_VEL
LIN {X 0,Y 29.632,Z 677.879,A -85,B 0,C 180,E1 -30978.415,E2 -30978.415} C_VEL
LIN {X 0,Y 18.396,Z 675.514,A -85,B 0,C 180,E1 -31000.16,E2 -31000.16} C_VEL
LIN {X 0,Y 14.872,Z 673.971,A -85,B 0,C 180,E1 -31021.785,E2 -31021.785} C_VEL
LIN {X 0,Y 13.824,Z 672.083,A -85,B 0,C 180,E1 -31049.987,E2 -31049.987} C_VEL
LIN {X 0,Y 16.278,Z 668.176,A -85,B 0,C 180,E1 -31090.347,E2 -31090.347} C_VEL
LIN {X 0,Y 26.57,Z 661.575,A -85,B 0,C 180,E1 -31117.768,E2 -31117.768} C_VEL
LIN {X 0,Y 38.247,Z 654.022,A -85,B 0,C 180,E1 -31128.305,E2 -31128.305} C_VEL
LIN {X 0,Y 49.502,Z 645.658,A -85,B 0,C 180,E1 -31133.597,E2 -31133.597} C_VEL
LIN {X 0,Y 61.567,Z 635.081,A -85,B 0,C 180,E1 -31137.167,E2 -31137.167} C_VEL
LIN {X 0,Y 71.896,Z 624.441,A -85,B 0,C 180,E1 -31139.122,E2 -31139.122} C_VEL
LIN {X 0,Y 81.437,Z 612.851,A -85,B 0,C 180,E1 -31140.492,E2 -31140.492} C_VEL
LIN {X 0,Y 90.513,Z 599.7,A -85,B 0,C 180,E1 -31141.495,E2 -31141.495} C_VEL
LIN {X 0,Y 98.464,Z 585.667,A -85,B 0,C 180,E1 -31142.245,E2 -31142.245} C_VEL
LIN {X 0,Y 105.097,Z 571.199,A -85,B 0,C 180,E1 -31142.735,E2 -31142.735} C_VEL
LIN {X 0,Y 110.634,Z 555.557,A -85,B 0,C 180,E1 -31143.135,E2 -31143.135} C_VEL
LIN {X 0,Y 114.437,Z 540.814,A -85,B 0,C 180,E1 -31143.413,E2 -31143.413} C_VEL
LIN {X 0,Y 118.15,Z 518.522,A -85,B 0,C 180,E1 -31143.779,E2 -31143.779} C_VEL
LIN {X 0,Y 118.893,Z 513.242,A -85,B 0,C 180,E1 -31143.943,E2 -31143.943} C_VEL
LIN {X 0,Y 117.737,Z 508.216,A -85,B 0,C 180,E1 -31148.063,E2 -31148.063} C_VEL
LIN {X 0,Y 117.208,Z 505.601,A -85,B 0,C 180,E1 -31150.816,E2 -31150.816} C_VEL
LIN {X 0,Y 116.711,Z 503.625,A -85,B 0,C 180,E1 -31153.939,E2 -31153.939} C_VEL
LIN {X 0,Y 116.413,Z 501.94,A -85,B 0,C 180,E1 -31157.57,E2 -31157.57} C_VEL
LIN {X 0,Y 116.331,Z 502.081,A -85,B 0,C 180,E1 -31162.46,E2 -31162.46} C_VEL
LIN {X 0,Y 116.842,Z 505.11,A -85,B 0,C 180,E1 -31168.765,E2 -31168.765} C_VEL
LIN {X 0,Y 117.669,Z 508.421,A -85,B 0,C 180,E1 -31172.976,E2 -31172.976} C_VEL
LIN {X 0,Y 118.693,Z 512.571,A -85,B 0,C 180,E1 -31176.675,E2 -31176.675} C_VEL
LIN {X 0,Y 115.166,Z 534.923,A -85,B 0,C 180,E1 -31177.102,E2 -31177.102} C_VEL
LIN {X 0,Y 113.094,Z 544.093,A -85,B 0,C 180,E1 -31177.31,E2 -31177.31} C_VEL
LIN {X 0,Y 111.422,Z 549.747,A -85,B 0,C 180,E1 -31177.076,E2 -31177.076} C_VEL
LIN {X 0,Y 104.888,Z 565.871,A -85,B 0,C 180,E1 -31174.883,E2 -31174.883} C_VEL
LIN {X 0,Y 102.5,Z 571.247,A -85,B 0,C 180,E1 -31174.499,E2 -31174.499} C_VEL
LIN {X 0,Y 101.7,Z 573.052,A -85,B 0,C 180,E1 -31174.508,E2 -31174.508} C_VEL
LIN {X 0,Y 94.453,Z 587.857,A -85,B 0,C 180,E1 -31175.071,E2 -31175.071} C_VEL
LIN {X 0,Y 86.499,Z 601.069,A -85,B 0,C 180,E1 -31175.664,E2 -31175.664} C_VEL
LIN {X 0,Y 77.577,Z 613.451,A -85,B 0,C 180,E1 -31176.488,E2 -31176.488} C_VEL
LIN {X 0,Y 67.339,Z 625.356,A -85,B 0,C 180,E1 -31177.627,E2 -31177.627} C_VEL
LIN {X 0,Y 56.984,Z 635.542,A -85,B 0,C 180,E1 -31179.076,E2 -31179.076} C_VEL
LIN {X 0,Y 46.607,Z 644.233,A -85,B 0,C 180,E1 -31181.071,E2 -31181.071} C_VEL
LIN {X 0,Y 34.556,Z 652.86,A -85,B 0,C 180,E1 -31184.624,E2 -31184.624} C_VEL
LIN {X 0,Y 22.46,Z 660.178,A -85,B 0,C 180,E1 -31191.268,E2 -31191.268} C_VEL
LIN {X 0,Y 10.608,Z 666.405,A -85,B 0,C 180,E1 -31210.672,E2 -31210.672} C_VEL
LIN {X 0,Y 7.169,Z 671.641,A -85,B 0,C 180,E1 -31308.734,E2 -31308.734} C_VEL
LIN {X 0,Y 14.137,Z 674.298,A -85,B 0,C 180,E1 -31337.723,E2 -31337.723} C_VEL
LIN {X 0,Y 11.055,Z 673.452,A -85,B 0,C 180,E1 -31350.352,E2 -31350.352} C_VEL
LIN {X 0,Y 6.736,Z 670.829,A -85,B 0,C 180,E1 -31409.973,E2 -31409.973} C_VEL
LIN {X 0,Y 11.781,Z 666.798,A -85,B 0,C 180,E1 -31473.45,E2 -31473.45} C_VEL
LIN {X 0,Y 24.768,Z 659.964,A -85,B 0,C 180,E1 -31493.225,E2 -31493.225} C_VEL
LIN {X 0,Y 37.094,Z 652.401,A -85,B 0,C 180,E1 -31498.972,E2 -31498.972} C_VEL
LIN {X 0,Y 49.221,Z 643.503,A -85,B 0,C 180,E1 -31501.933,E2 -31501.933} C_VEL
LIN {X 0,Y 59.854,Z 634.231,A -85,B 0,C 180,E1 -31503.619,E2 -31503.619} C_VEL
LIN {X 0,Y 70.511,Z 623.343,A -85,B 0,C 180,E1 -31504.674,E2 -31504.674} C_VEL
LIN {X 0,Y 80.297,Z 611.464,A -85,B 0,C 180,E1 -31505.401,E2 -31505.401} C_VEL
LIN {X 0,Y 89.199,Z 598.531,A -85,B 0,C 180,E1 -31505.907,E2 -31505.907} C_VEL
LIN {X 0,Y 97.216,Z 584.349,A -85,B 0,C 180,E1 -31506.284,E2 -31506.284} C_VEL
LIN {X 0,Y 103.895,Z 569.627,A -85,B 0,C 180,E1 -31506.535,E2 -31506.535} C_VEL
LIN {X 0,Y 109.241,Z 554.371,A -85,B 0,C 180,E1 -31506.718,E2 -31506.718} C_VEL
LIN {X 0,Y 113.049,Z 539.32,A -85,B 0,C 180,E1 -31506.92,E2 -31506.92} C_VEL
LIN {X 0,Y 116.703,Z 517.043,A -85,B 0,C 180,E1 -31507.225,E2 -31507.225} C_VEL
LIN {X 0,Y 115.939,Z 512.405,A -85,B 0,C 180,E1 -31511.622,E2 -31511.622} C_VEL
LIN {X 0,Y 115.483,Z 510.373,A -85,B 0,C 180,E1 -31514.896,E2 -31514.896} C_VEL
LIN {X 0,Y 115.303,Z 509.101,A -85,B 0,C 180,E1 -31517.745,E2 -31517.745} C_VEL
LIN {X 0,Y 115.258,Z 508.965,A -85,B 0,C 180,E1 -31521.765,E2 -31521.765} C_VEL
LIN {X 0,Y 115.599,Z 511.978,A -85,B 0,C 180,E1 -31528.033,E2 -31528.033} C_VEL
LIN {X 0,Y 116.315,Z 515.401,A -85,B 0,C 180,E1 -31532.234,E2 -31532.234} C_VEL
LIN {X 0,Y 116.561,Z 516.613,A -85,B 0,C 180,E1 -31533.402,E2 -31533.402} C_VEL
LIN {X 0,Y 113.373,Z 535.984,A -85,B 0,C 180,E1 -31533.646,E2 -31533.646} C_VEL
LIN {X 0,Y 109.62,Z 551.204,A -85,B 0,C 180,E1 -31533.96,E2 -31533.96} C_VEL
LIN {X 0,Y 104.736,Z 565.654,A -85,B 0,C 180,E1 -31534.293,E2 -31534.293} C_VEL
LIN {X 0,Y 101.7,Z 573.052,A -85,B 0,C 180,E1 -31534.508,E2 -31534.508} C_VEL
LIN {X 0,Y 99.156,Z 578.375,A -85,B 0,C 180,E1 -31534.3,E2 -31534.3} C_VEL
LIN {X 0,Y 94.448,Z 586.792,A -85,B 0,C 180,E1 -31532.929,E2 -31532.929} C_VEL
LIN {X 0,Y 89.336,Z 594.947,A -85,B 0,C 180,E1 -31531.369,E2 -31531.369} C_VEL
LIN {X 0,Y 86.073,Z 599.866,A -85,B 0,C 180,E1 -31530.993,E2 -31530.993} C_VEL
LIN {X 0,Y 76.269,Z 613.493,A -85,B 0,C 180,E1 -31531.281,E2 -31531.281} C_VEL
LIN {X 0,Y 66.023,Z 625.352,A -85,B 0,C 180,E1 -31531.621,E2 -31531.621} C_VEL
LIN {X 0,Y 54.574,Z 636.469,A -85,B 0,C 180,E1 -31532.057,E2 -31532.057} C_VEL
LIN {X 0,Y 41.677,Z 646.879,A -85,B 0,C 180,E1 -31532.534,E2 -31532.534} C_VEL
LIN {X 0,Y 29.629,Z 655.009,A -85,B 0,C 180,E1 -31532.869,E2 -31532.869} C_VEL
LIN {X 0,Y 16.644,Z 662.253,A -85,B 0,C 180,E1 -31532.404,E2 -31532.404} C_VEL
LIN {X 0,Y 6.039,Z 667.167,A -85,B 0,C 180,E1 -31524.907,E2 -31524.907} C_VEL
LIN {X 0,Y 7.147,Z 666.832,A -85,B 0,C 180,E1 -31510.596,E2 -31510.596} C_VEL
LIN {X 0,Y 21.383,Z 660.145,A -85,B 0,C 180,E1 -31509.645,E2 -31509.645} C_VEL
LIN {X 0,Y 33.879,Z 652.838,A -85,B 0,C 180,E1 -31509.847,E2 -31509.847} C_VEL
LIN {X 0,Y 46.394,Z 644.001,A -85,B 0,C 180,E1 -31510.073,E2 -31510.073} C_VEL
LIN {X 0,Y 57.151,Z 634.927,A -85,B 0,C 180,E1 -31510.351,E2 -31510.351} C_VEL
LIN {X 0,Y 67.869,Z 624.304,A -85,B 0,C 180,E1 -31510.358,E2 -31510.358} C_VEL
LIN {X 0,Y 77.753,Z 612.655,A -85,B 0,C 180,E1 -31510.417,E2 -31510.417} C_VEL
LIN {X 0,Y 86.636,Z 600.182,A -85,B 0,C 180,E1 -31510.404,E2 -31510.404} C_VEL
LIN {X 0,Y 94.688,Z 586.443,A -85,B 0,C 180,E1 -31510.45,E2 -31510.45} C_VEL
LIN {X 0,Y 101.383,Z 572.355,A -85,B 0,C 180,E1 -31510.434,E2 -31510.434} C_VEL
LIN {X 0,Y 106.298,Z 559.464,A -85,B 0,C 180,E1 -31510.439,E2 -31510.439} C_VEL
LIN {X 0,Y 110.625,Z 544.538,A -85,B 0,C 180,E1 -31510.423,E2 -31510.423} C_VEL
LIN {X 0,Y 113.771,Z 528.392,A -85,B 0,C 180,E1 -31510.541,E2 -31510.541} C_VEL
LIN {X 0,Y 114.849,Z 521.108,A -85,B 0,C 180,E1 -31510.695,E2 -31510.695} C_VEL
LIN {X 0,Y 114.553,Z 518.629,A -85,B 0,C 180,E1 -31513.284,E2 -31513.284} C_VEL
LIN {X 0,Y 114.258,Z 516.947,A -85,B 0,C 180,E1 -31516.284,E2 -31516.284} C_VEL
LIN {X 0,Y 114.2,Z 516.221,A -85,B 0,C 180,E1 -31517.922,E2 -31517.922} C_VEL
LIN {X 0,Y 114.144,Z 516.291,A -85,B 0,C 180,E1 -31521.989,E2 -31521.989} C_VEL
LIN {X 0,Y 114.374,Z 518.802,A -85,B 0,C 180,E1 -31527.249,E2 -31527.249} C_VEL
LIN {X 0,Y 114.74,Z 521.006,A -85,B 0,C 180,E1 -31529.986,E2 -31529.986} C_VEL
LIN {X 0,Y 111.53,Z 539.087,A -85,B 0,C 180,E1 -31530.108,E2 -31530.108} C_VEL
LIN {X 0,Y 107.36,Z 554.726,A -85,B 0,C 180,E1 -31530.313,E2 -31530.313} C_VEL
LIN {X 0,Y 101.961,Z 569.6,A -85,B 0,C 180,E1 -31530.506,E2 -31530.506} C_VEL
LIN {X 0,Y 95.273,Z 584.015,A -85,B 0,C 180,E1 -31530.725,E2 -31530.725} C_VEL
LIN {X 0,Y 88.089,Z 596.644,A -85,B 0,C 180,E1 -31530.948,E2 -31530.948} C_VEL
LIN {X 0,Y 86.073,Z 599.866,A -85,B 0,C 180,E1 -31530.993,E2 -31530.993} C_VEL
LIN {X 0,Y 82.675,Z 604.738,A -85,B 0,C 180,E1 -31530.598,E2 -31530.598} C_VEL
LIN {X 0,Y 76.807,Z 612.265,A -85,B 0,C 180,E1 -31528.65,E2 -31528.65} C_VEL
LIN {X 0,Y 70.733,Z 619.478,A -85,B 0,C 180,E1 -31526.347,E2 -31526.347} C_VEL
LIN {X 0,Y 66.832,Z 623.804,A -85,B 0,C 180,E1 -31525.557,E2 -31525.557} C_VEL
LIN {X 0,Y 56.096,Z 634.6,A -85,B 0,C 180,E1 -31524.734,E2 -31524.734} C_VEL
LIN {X 0,Y 45.985,Z 643.291,A -85,B 0,C 180,E1 -31523.52,E2 -31523.52} C_VEL
LIN {X 0,Y 37.68,Z 649.522,A -85,B 0,C 180,E1 -31521.907,E2 -31521.907} C_VEL
LIN {X 0,Y 37.56,Z 649.636,A -85,B 0,C 180,E1 -31520.693,E2 -31520.693} C_VEL
LIN {X 0,Y 48.168,Z 641.72,A -85,B 0,C 180,E1 -31518.5,E2 -31518.5} C_VEL
LIN {X 0,Y 58.847,Z 632.316,A -85,B 0,C 180,E1 -31517.181,E2 -31517.181} C_VEL
LIN {X 0,Y 70.403,Z 620.264,A -85,B 0,C 180,E1 -31516.101,E2 -31516.101} C_VEL
LIN {X 0,Y 80.19,Z 607.99,A -85,B 0,C 180,E1 -31515.416,E2 -31515.416} C_VEL
LIN {X 0,Y 89.09,Z 594.534,A -85,B 0,C 180,E1 -31514.913,E2 -31514.913} C_VEL
LIN {X 0,Y 96.228,Z 581.418,A -85,B 0,C 180,E1 -31514.607,E2 -31514.607} C_VEL
LIN {X 0,Y 102.886,Z 566.206,A -85,B 0,C 180,E1 -31514.281,E2 -31514.281} C_VEL
LIN {X 0,Y 108.019,Z 550.76,A -85,B 0,C 180,E1 -31514.114,E2 -31514.114} C_VEL
LIN {X 0,Y 111.663,Z 535.357,A -85,B 0,C 180,E1 -31514.086,E2 -31514.086} C_VEL
LIN {X 0,Y 113.317,Z 525.44,A -85,B 0,C 180,E1 -31514.137,E2 -31514.137} C_VEL
LIN {X 0,Y 113.12,Z 523.767,A -85,B 0,C 180,E1 -31517.087,E2 -31517.087} C_VEL
LIN {X 0,Y 113.098,Z 523.342,A -85,B 0,C 180,E1 -31518.103,E2 -31518.103} C_VEL
LIN {X 0,Y 113.065,Z 523.299,A -85,B 0,C 180,E1 -31521.547,E2 -31521.547} C_VEL
LIN {X 0,Y 113.164,Z 525.639,A -85,B 0,C 180,E1 -31526.42,E2 -31526.42} C_VEL
LIN {X 0,Y 110.153,Z 541.523,A -85,B 0,C 180,E1 -31526.484,E2 -31526.484} C_VEL
LIN {X 0,Y 105.939,Z 556.657,A -85,B 0,C 180,E1 -31526.566,E2 -31526.566} C_VEL
LIN {X 0,Y 100.134,Z 572.12,A -85,B 0,C 180,E1 -31526.513,E2 -31526.513} C_VEL
LIN {X 0,Y 93.217,Z 586.539,A -85,B 0,C 180,E1 -31526.457,E2 -31526.457} C_VEL
LIN {X 0,Y 85.24,Z 600.036,A -85,B 0,C 180,E1 -31526.262,E2 -31526.262} C_VEL
LIN {X 0,Y 75.221,Z 613.984,A -85,B 0,C 180,E1 -31525.943,E2 -31525.943} C_VEL
LIN {X 0,Y 66.832,Z 623.804,A -85,B 0,C 180,E1 -31525.557,E2 -31525.557} C_VEL
LIN {X 0,Y 67.204,Z 623.37,A -85,B 0,C 180,E1 -31524.74,E2 -31524.74} C_VEL
LIN {X 0,Y 67.89,Z 622.598,A -85,B 0,C 180,E1 -31524.215,E2 -31524.215} C_VEL
LIN {X 0,Y 72.459,Z 617.273,A -85,B 0,C 180,E1 -31522.632,E2 -31522.632} C_VEL
LIN {X 0,Y 78.883,Z 609.042,A -85,B 0,C 180,E1 -31521.64,E2 -31521.64} C_VEL
LIN {X 0,Y 84.06,Z 601.624,A -85,B 0,C 180,E1 -31521.433,E2 -31521.433} C_VEL
LIN {X 0,Y 85.68,Z 599.082,A -85,B 0,C 180,E1 -31521.538,E2 -31521.538} C_VEL
LIN {X 0,Y 93.379,Z 585.763,A -85,B 0,C 180,E1 -31522.107,E2 -31522.107} C_VEL
LIN {X 0,Y 100.241,Z 571.118,A -85,B 0,C 180,E1 -31522.476,E2 -31522.476} C_VEL
LIN {X 0,Y 105.765,Z 556.066,A -85,B 0,C 180,E1 -31522.731,E2 -31522.731} C_VEL
LIN {X 0,Y 109.875,Z 541.001,A -85,B 0,C 180,E1 -31522.787,E2 -31522.787} C_VEL
LIN {X 0,Y 111.834,Z 531.182,A -85,B 0,C 180,E1 -31522.853,E2 -31522.853} C_VEL
LIN {X 0,Y 111.955,Z 530.196,A -85,B 0,C 180,E1 -31520.922,E2 -31520.922} C_VEL
LIN {X 0,Y 111.962,Z 530.67,A -85,B 0,C 180,E1 -31517.704,E2 -31517.704} C_VEL
LIN {X 0,Y 108.53,Z 546.774,A -85,B 0,C 180,E1 -31517.806,E2 -31517.806} C_VEL
LIN {X 0,Y 104.164,Z 561.113,A -85,B 0,C 180,E1 -31518.122,E2 -31518.122} C_VEL
LIN {X 0,Y 99.142,Z 573.959,A -85,B 0,C 180,E1 -31518.54,E2 -31518.54} C_VEL
LIN {X 0,Y 92.171,Z 588.19,A -85,B 0,C 180,E1 -31519.176,E2 -31519.176} C_VEL
LIN {X 0,Y 84.127,Z 601.584,A -85,B 0,C 180,E1 -31519.983,E2 -31519.983} C_VEL
LIN {X 0,Y 79.688,Z 608.001,A -85,B 0,C 180,E1 -31520.525,E2 -31520.525} C_VEL
LIN {X 0,Y 78.754,Z 609.231,A -85,B 0,C 180,E1 -31520.916,E2 -31520.916} C_VEL
LIN {X 0,Y 85.68,Z 599.082,A -85,B 0,C 180,E1 -31521.538,E2 -31521.538} C_VEL
LIN {X 0,Y 89.337,Z 600.146,A -85,B 0,C 180,E1 -31521.878,E2 -31521.878} C_VEL
LIN {X 0,Y 89.337,Z 600.146,A -85,B 0,C 180,E1 -31521.878,E2 -31521.878}

QRS_NEXT_CUT()

QRS_NEXT()
QRS_HOME()

END
